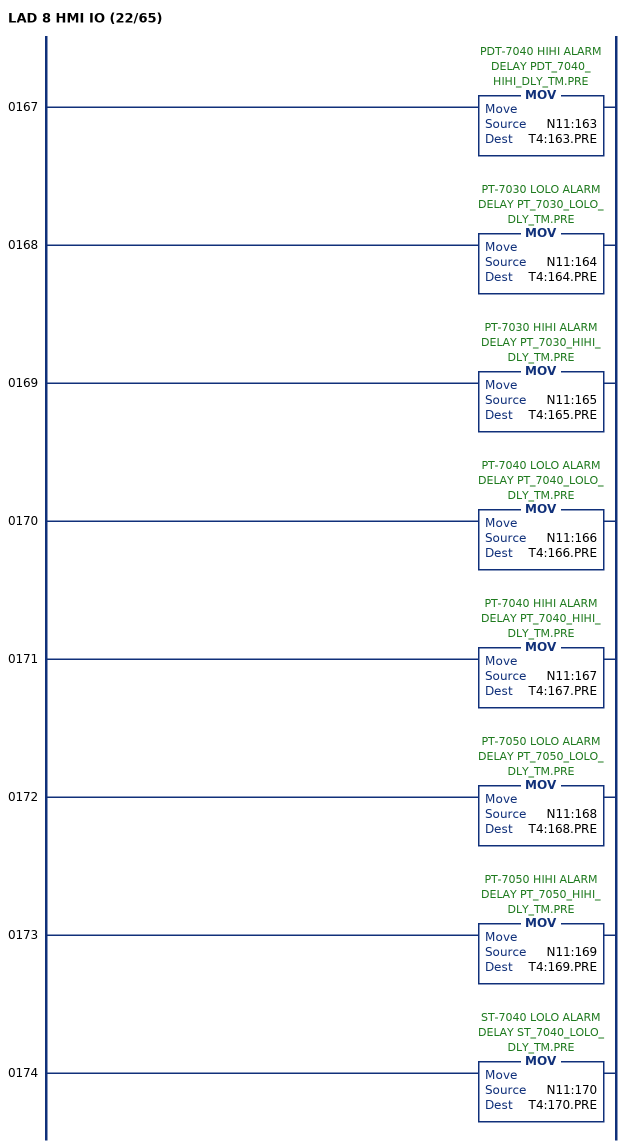
% Rung: 167 %
SOR MOV N11:163 T4:163.PRE EOR
%   N11:163  PDT_7040_HIHI_DLY_SP  "PDT-7040 HIHI ALARM DELAY SP FROM HMI" %
%   T4:163  PDT_7040_HIHI_DLY_TM  "PDT-7040 HIHI ALARM DELAY" %
% Rung: 168 %
SOR MOV N11:164 T4:164.PRE EOR
%   N11:164  PT_7030_LOLO_DLY_SP  "PT-7030 LOLO ALARM DELAY SP FROM HMI" %
%   T4:164  PT_7030_LOLO_DLY_TM  "PT-7030 LOLO ALARM DELAY" %
% Rung: 169 %
SOR MOV N11:165 T4:165.PRE EOR
%   N11:165  PT_7030_HIHI_DLY_SP  "PT-7030 HIHI ALARM DELAY SP FROM HMI" %
%   T4:165  PT_7030_HIHI_DLY_TM  "PT-7030 HIHI ALARM DELAY" %
% Rung: 170 %
SOR MOV N11:166 T4:166.PRE EOR
%   N11:166  PT_7040_LOLO_DLY_SP  "PT-7040 LOLO ALARM DELAY SP FROM HMI" %
%   T4:166  PT_7040_LOLO_DLY_TM  "PT-7040 LOLO ALARM DELAY" %
% Rung: 171 %
SOR MOV N11:167 T4:167.PRE EOR
%   N11:167  PT_7040_HIHI_DLY_SP  "PT-7040 HIHI ALARM DELAY SP FROM HMI" %
%   T4:167  PT_7040_HIHI_DLY_TM  "PT-7040 HIHI ALARM DELAY" %
% Rung: 172 %
SOR MOV N11:168 T4:168.PRE EOR
%   N11:168  PT_7050_LOLO_DLY_SP  "PT-7050 LOLO ALARM DELAY SP FROM HMI" %
%   T4:168  PT_7050_LOLO_DLY_TM  "PT-7050 LOLO ALARM DELAY" %
% Rung: 173 %
SOR MOV N11:169 T4:169.PRE EOR
%   N11:169  PT_7050_HIHI_DLY_SP  "PT-7050 HIHI ALARM DELAY SP FROM HMI" %
%   T4:169  PT_7050_HIHI_DLY_TM  "PT-7050 HIHI ALARM DELAY" %
% Rung: 174 %
SOR MOV N11:170 T4:170.PRE EOR
%   N11:170  ST_7040_LOLO_DLY_SP  "ST-7040 LOLO ALARM DELAY SP FROM HMI" %
%   T4:170  ST_7040_LOLO_DLY_TM  "ST-7040 LOLO ALARM DELAY" %

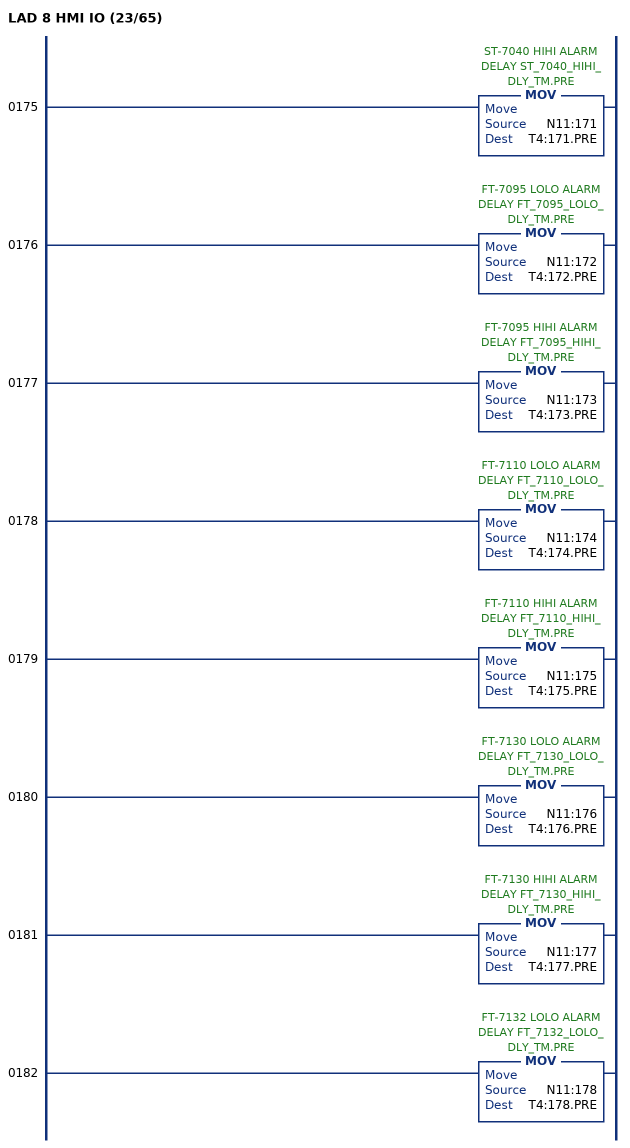
% Rung: 175 %
SOR MOV N11:171 T4:171.PRE EOR
%   N11:171  ST_7040_HIHI_DLY_SP  "ST-7040 HIHI ALARM DELAY SP FROM HMI" %
%   T4:171  ST_7040_HIHI_DLY_TM  "ST-7040 HIHI ALARM DELAY" %
% Rung: 176 %
SOR MOV N11:172 T4:172.PRE EOR
%   N11:172  FT_7095_LOLO_DLY_SP  "FT-7095 LOLO ALARM DELAY SP FROM HMI" %
%   T4:172  FT_7095_LOLO_DLY_TM  "FT-7095 LOLO ALARM DELAY" %
% Rung: 177 %
SOR MOV N11:173 T4:173.PRE EOR
%   N11:173  FT_7095_HIHI_DLY_SP  "FT-7095 HIHI ALARM DELAY SP FROM HMI" %
%   T4:173  FT_7095_HIHI_DLY_TM  "FT-7095 HIHI ALARM DELAY" %
% Rung: 178 %
SOR MOV N11:174 T4:174.PRE EOR
%   N11:174  FT_7110_LOLO_DLY_SP  "FT-7110 LOLO ALARM DELAY SP FROM HMI" %
%   T4:174  FT_7110_LOLO_DLY_TM  "FT-7110 LOLO ALARM DELAY" %
% Rung: 179 %
SOR MOV N11:175 T4:175.PRE EOR
%   N11:175  FT_7110_HIHI_DLY_SP  "FT-7110 HIHI ALARM DELAY SP FROM HMI" %
%   T4:175  FT_7110_HIHI_DLY_TM  "FT-7110 HIHI ALARM DELAY" %
% Rung: 180 %
SOR MOV N11:176 T4:176.PRE EOR
%   N11:176  FT_7130_LOLO_DLY_SP  "FT-7130 LOLO ALARM DELAY SP FROM HMI" %
%   T4:176  FT_7130_LOLO_DLY_TM  "FT-7130 LOLO ALARM DELAY" %
% Rung: 181 %
SOR MOV N11:177 T4:177.PRE EOR
%   N11:177  FT_7130_HIHI_DLY_SP  "FT-7130 HIHI ALARM DELAY SP FROM HMI" %
%   T4:177  FT_7130_HIHI_DLY_TM  "FT-7130 HIHI ALARM DELAY" %
% Rung: 182 %
SOR MOV N11:178 T4:178.PRE EOR
%   N11:178  FT_7132_LOLO_DLY_SP  "FT-7132 LOLO ALARM DELAY SP FROM HMI" %
%   T4:178  FT_7132_LOLO_DLY_TM  "FT-7132 LOLO ALARM DELAY" %

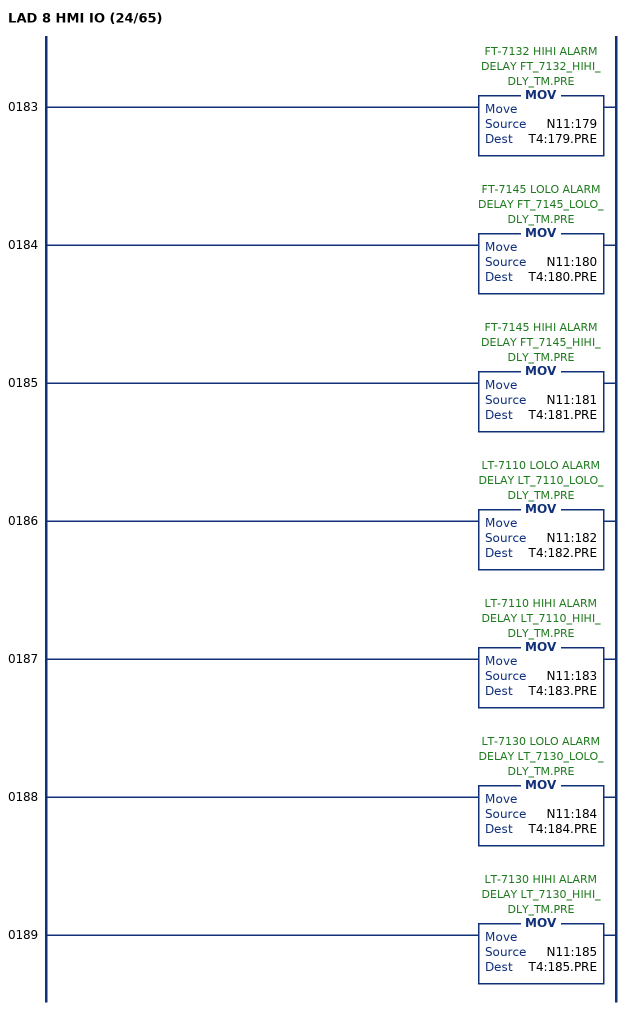
% Rung: 183 %
SOR MOV N11:179 T4:179.PRE EOR
%   N11:179  FT_7132_HIHI_DLY_SP  "FT-7132 HIHI ALARM DELAY SP FROM HMI" %
%   T4:179  FT_7132_HIHI_DLY_TM  "FT-7132 HIHI ALARM DELAY" %
% Rung: 184 %
SOR MOV N11:180 T4:180.PRE EOR
%   N11:180  FT_7145_LOLO_DLY_SP  "FT-7145 LOLO ALARM DELAY SP FROM HMI" %
%   T4:180  FT_7145_LOLO_DLY_TM  "FT-7145 LOLO ALARM DELAY" %
% Rung: 185 %
SOR MOV N11:181 T4:181.PRE EOR
%   N11:181  FT_7145_HIHI_DLY_SP  "FT-7145 HIHI ALARM DELAY SP FROM HMI" %
%   T4:181  FT_7145_HIHI_DLY_TM  "FT-7145 HIHI ALARM DELAY" %
% Rung: 186 %
SOR MOV N11:182 T4:182.PRE EOR
%   N11:182  LT_7110_LOLO_DLY_SP  "LT-7110 LOLO ALARM DELAY SP FROM HMI" %
%   T4:182  LT_7110_LOLO_DLY_TM  "LT-7110 LOLO ALARM DELAY" %
% Rung: 187 %
SOR MOV N11:183 T4:183.PRE EOR
%   N11:183  LT_7110_HIHI_DLY_SP  "LT-7110 HIHI ALARM DELAY SP FROM HMI" %
%   T4:183  LT_7110_HIHI_DLY_TM  "LT-7110 HIHI ALARM DELAY" %
% Rung: 188 %
SOR MOV N11:184 T4:184.PRE EOR
%   N11:184  LT_7130_LOLO_DLY_SP  "LT-7130 LOLO ALARM DELAY SP FROM HMI" %
%   T4:184  LT_7130_LOLO_DLY_TM  "LT-7130 LOLO ALARM DELAY" %
% Rung: 189 %
SOR MOV N11:185 T4:185.PRE EOR
%   N11:185  LT_7130_HIHI_DLY_SP  "LT-7130 HIHI ALARM DELAY SP FROM HMI" %
%   T4:185  LT_7130_HIHI_DLY_TM  "LT-7130 HIHI ALARM DELAY" %

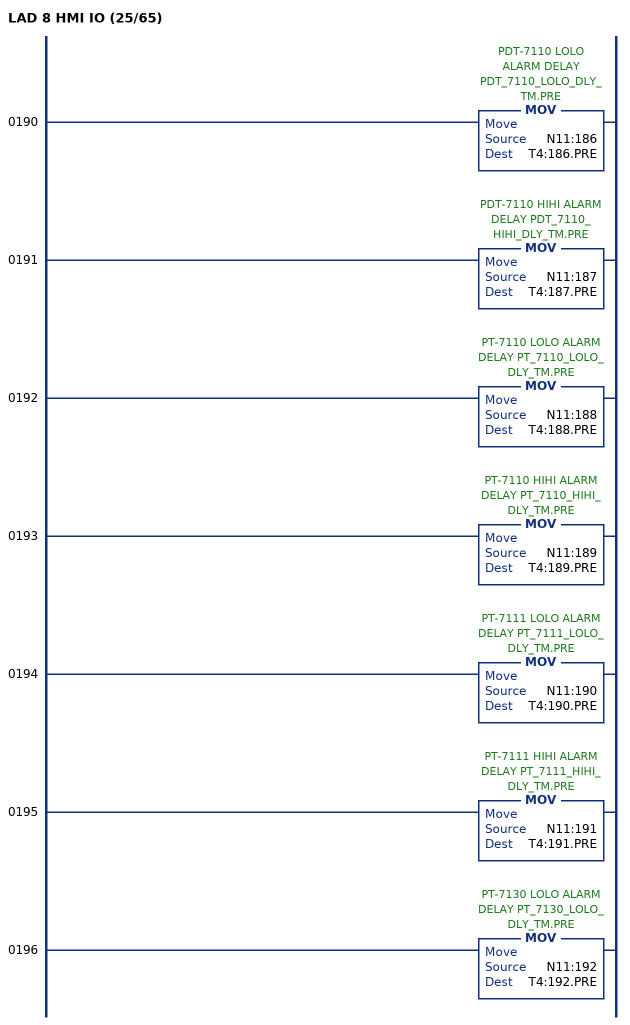
% Rung: 190 %
SOR MOV N11:186 T4:186.PRE EOR
%   N11:186  PDT_7110_LOLO_DLY_SP  "PDT-7110 LOLO ALARM DELAY SP FROM HMI" %
%   T4:186  PDT_7110_LOLO_DLY_TM  "PDT-7110 LOLO ALARM DELAY" %
% Rung: 191 %
SOR MOV N11:187 T4:187.PRE EOR
%   N11:187  PDT_7110_HIHI_DLY_SP  "PDT-7110 HIHI ALARM DELAY SP FROM HMI" %
%   T4:187  PDT_7110_HIHI_DLY_TM  "PDT-7110 HIHI ALARM DELAY" %
% Rung: 192 %
SOR MOV N11:188 T4:188.PRE EOR
%   N11:188  PT_7110_LOLO_DLY_SP  "PT-7110 LOLO ALARM DELAY SP FROM HMI" %
%   T4:188  PT_7110_LOLO_DLY_TM  "PT-7110 LOLO ALARM DELAY" %
% Rung: 193 %
SOR MOV N11:189 T4:189.PRE EOR
%   N11:189  PT_7110_HIHI_DLY_SP  "PT-7110 HIHI ALARM DELAY SP FROM HMI" %
%   T4:189  PT_7110_HIHI_DLY_TM  "PT-7110 HIHI ALARM DELAY" %
% Rung: 194 %
SOR MOV N11:190 T4:190.PRE EOR
%   N11:190  PT_7111_LOLO_DLY_SP  "PT-7111 LOLO ALARM DELAY SP FROM HMI" %
%   T4:190  PT_7111_LOLO_DLY_TM  "PT-7111 LOLO ALARM DELAY" %
% Rung: 195 %
SOR MOV N11:191 T4:191.PRE EOR
%   N11:191  PT_7111_HIHI_DLY_SP  "PT-7111 HIHI ALARM DELAY SP FROM HMI" %
%   T4:191  PT_7111_HIHI_DLY_TM  "PT-7111 HIHI ALARM DELAY" %
% Rung: 196 %
SOR MOV N11:192 T4:192.PRE EOR
%   N11:192  PT_7130_LOLO_DLY_SP  "PT-7130 LOLO ALARM DELAY SP FROM HMI" %
%   T4:192  PT_7130_LOLO_DLY_TM  "PT-7130 LOLO ALARM DELAY" %

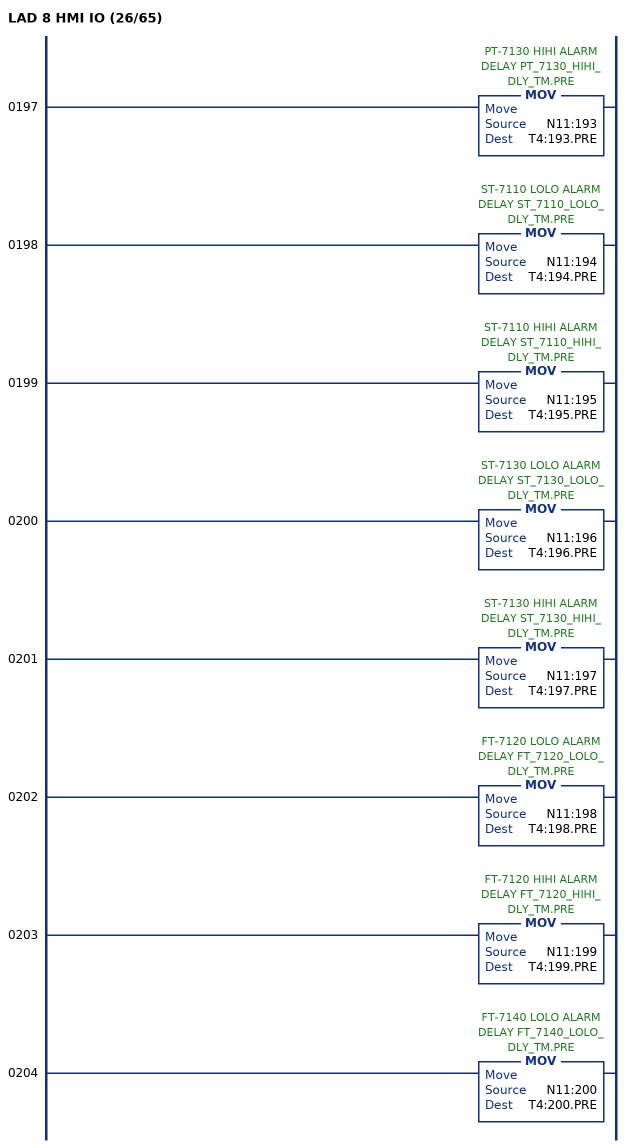
% Rung: 197 %
SOR MOV N11:193 T4:193.PRE EOR
%   N11:193  PT_7130_HIHI_DLY_SP  "PT-7130 HIHI ALARM DELAY SP FROM HMI" %
%   T4:193  PT_7130_HIHI_DLY_TM  "PT-7130 HIHI ALARM DELAY" %
% Rung: 198 %
SOR MOV N11:194 T4:194.PRE EOR
%   N11:194  ST_7110_LOLO_DLY_SP  "ST-7110 LOLO ALARM DELAY SP FROM HMI" %
%   T4:194  ST_7110_LOLO_DLY_TM  "ST-7110 LOLO ALARM DELAY" %
% Rung: 199 %
SOR MOV N11:195 T4:195.PRE EOR
%   N11:195  ST_7110_HIHI_DLY_SP  "ST-7110 HIHI ALARM DELAY SP FROM HMI" %
%   T4:195  ST_7110_HIHI_DLY_TM  "ST-7110 HIHI ALARM DELAY" %
% Rung: 200 %
SOR MOV N11:196 T4:196.PRE EOR
%   N11:196  ST_7130_LOLO_DLY_SP  "ST-7130 LOLO ALARM DELAY SP FROM HMI" %
%   T4:196  ST_7130_LOLO_DLY_TM  "ST-7130 LOLO ALARM DELAY" %
% Rung: 201 %
SOR MOV N11:197 T4:197.PRE EOR
%   N11:197  ST_7130_HIHI_DLY_SP  "ST-7130 HIHI ALARM DELAY SP FROM HMI" %
%   T4:197  ST_7130_HIHI_DLY_TM  "ST-7130 HIHI ALARM DELAY" %
% Rung: 202 %
SOR MOV N11:198 T4:198.PRE EOR
%   N11:198  FT_7120_LOLO_DLY_SP  "FT-7120 LOLO ALARM DELAY SP FROM HMI" %
%   T4:198  FT_7120_LOLO_DLY_TM  "FT-7120 LOLO ALARM DELAY" %
% Rung: 203 %
SOR MOV N11:199 T4:199.PRE EOR
%   N11:199  FT_7120_HIHI_DLY_SP  "FT-7120 HIHI ALARM DELAY SP FROM HMI" %
%   T4:199  FT_7120_HIHI_DLY_TM  "FT-7120 HIHI ALARM DELAY" %
% Rung: 204 %
SOR MOV N11:200 T4:200.PRE EOR
%   N11:200  FT_7140_LOLO_DLY_SP  "FT-7140 LOLO ALARM DELAY SP FROM HMI" %
%   T4:200  FT_7140_LOLO_DLY_TM  "FT-7140 LOLO ALARM DELAY" %

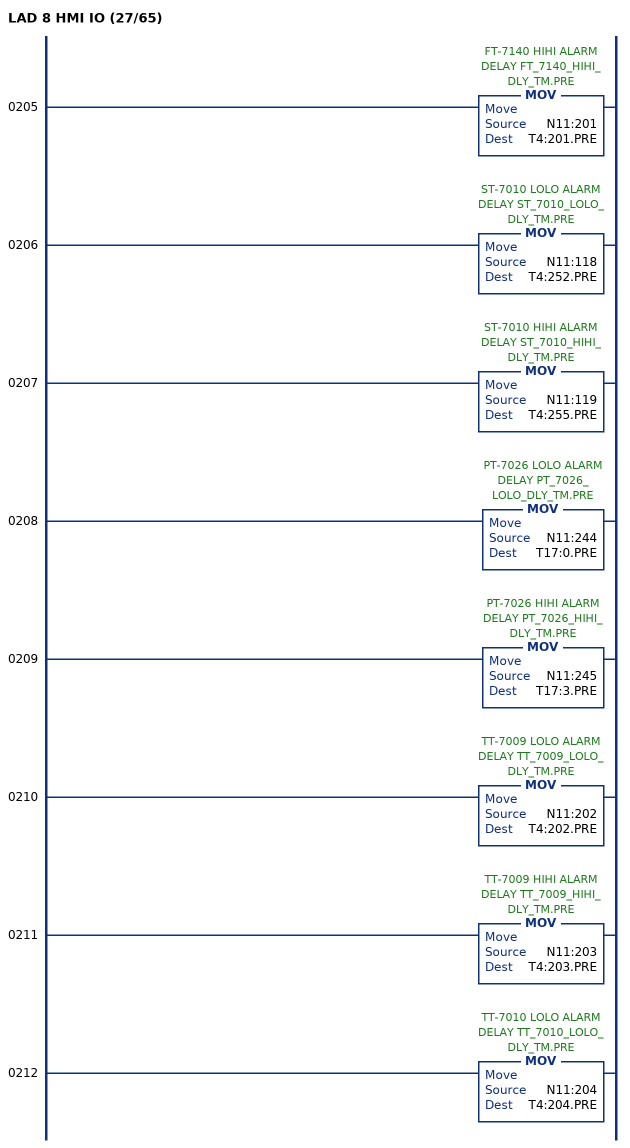
% Rung: 205 %
SOR MOV N11:201 T4:201.PRE EOR
%   N11:201  FT_7140_HIHI_DLY_SP  "FT-7140 HIHI ALARM DELAY SP FROM HMI" %
%   T4:201  FT_7140_HIHI_DLY_TM  "FT-7140 HIHI ALARM DELAY" %
% Rung: 206 %
SOR MOV N11:118 T4:252.PRE EOR
%   N11:118  ST_7010_LOLO_DLY_SP  "ST-7010 LL ALARM DELAY SP FROM HMI" %
%   T4:252  ST_7010_LOLO_DLY_TM  "ST-7010 LOLO ALARM DELAY" %
% Rung: 207 %
SOR MOV N11:119 T4:255.PRE EOR
%   N11:119  ST_7010_HIHI_DLY_SP  "ST-7010 HH ALARM DELAY SP FROM HMI" %
%   T4:255  ST_7010_HIHI_DLY_TM  "ST-7010 HIHI ALARM DELAY" %
% Rung: 208 %
SOR MOV N11:244 T17:0.PRE EOR
%   N11:244  PT_7026_LOLO_DLY_SP  "PT-7026 LL ALARM DELAY SP FROM HMI" %
%   T17:0  PT_7026_LOLO_DLY_TM  "PT-7026 LOLO ALARM DELAY" %
% Rung: 209 %
SOR MOV N11:245 T17:3.PRE EOR
%   N11:245  PT_7026_HIHI_DLY_SP  "PT-7026 HH ALARM DELAY SP FROM HMI" %
%   T17:3  PT_7026_HIHI_DLY_TM  "PT-7026 HIHI ALARM DELAY" %
% Rung: 210 %
SOR MOV N11:202 T4:202.PRE EOR
%   N11:202  TT_7009_LOLO_DLY_SP  "TT-7009 LOLO ALARM DELAY SP FROM HMI" %
%   T4:202  TT_7009_LOLO_DLY_TM  "TT-7009 LOLO ALARM DELAY" %
% Rung: 211 %
SOR MOV N11:203 T4:203.PRE EOR
%   N11:203  TT_7009_HIHI_DLY_SP  "TT-7009 HIHI ALARM DELAY SP FROM HMI" %
%   T4:203  TT_7009_HIHI_DLY_TM  "TT-7009 HIHI ALARM DELAY" %
% Rung: 212 %
SOR MOV N11:204 T4:204.PRE EOR
%   N11:204  TT_7010_LOLO_DLY_SP  "TT-7010 LOLO ALARM DELAY SP FROM HMI" %
%   T4:204  TT_7010_LOLO_DLY_TM  "TT-7010 LOLO ALARM DELAY" %

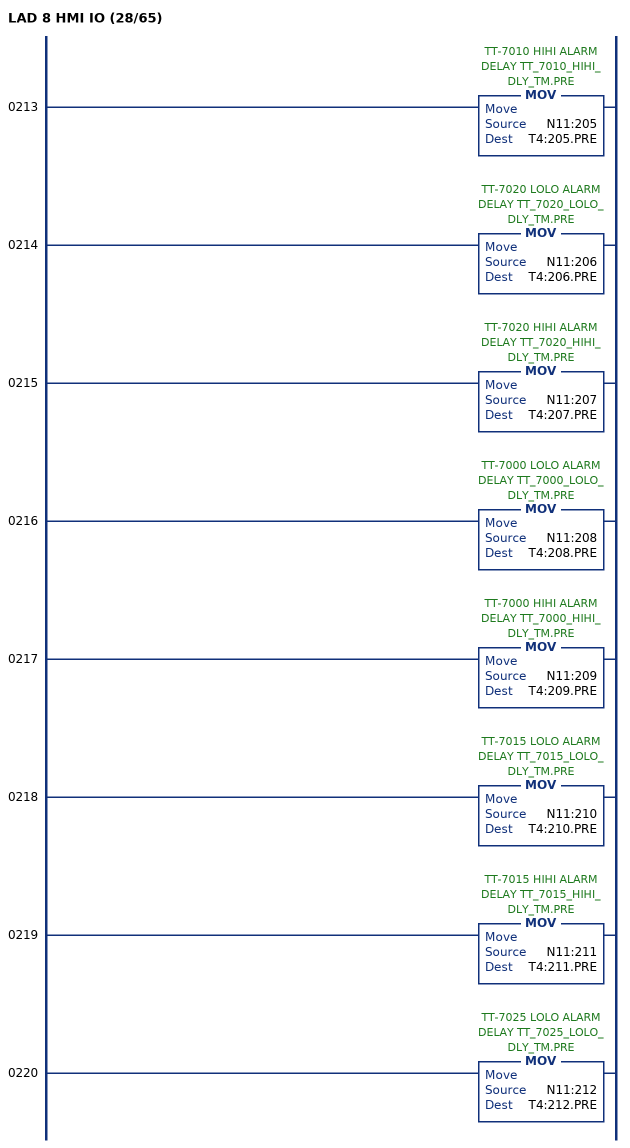
% Rung: 213 %
SOR MOV N11:205 T4:205.PRE EOR
%   N11:205  TT_7010_HIHI_DLY_SP  "TT-7010 HIHI ALARM DELAY SP FROM HMI" %
%   T4:205  TT_7010_HIHI_DLY_TM  "TT-7010 HIHI ALARM DELAY" %
% Rung: 214 %
SOR MOV N11:206 T4:206.PRE EOR
%   N11:206  TT_7020_LOLO_DLY_SP  "TT-7020 LOLO ALARM DELAY SP FROM HMI" %
%   T4:206  TT_7020_LOLO_DLY_TM  "TT-7020 LOLO ALARM DELAY" %
% Rung: 215 %
SOR MOV N11:207 T4:207.PRE EOR
%   N11:207  TT_7020_HIHI_DLY_SP  "TT-7020 HIHI ALARM DELAY SP FROM HMI" %
%   T4:207  TT_7020_HIHI_DLY_TM  "TT-7020 HIHI ALARM DELAY" %
% Rung: 216 %
SOR MOV N11:208 T4:208.PRE EOR
%   N11:208  TT_7000_LOLO_DLY_SP  "TT-7000 LOLO ALARM DELAY SP FROM HMI" %
%   T4:208  TT_7000_LOLO_DLY_TM  "TT-7000 LOLO ALARM DELAY" %
% Rung: 217 %
SOR MOV N11:209 T4:209.PRE EOR
%   N11:209  TT_7000_HIHI_DLY_SP  "TT-7000 HIHI ALARM DELAY SP FROM HMI" %
%   T4:209  TT_7000_HIHI_DLY_TM  "TT-7000 HIHI ALARM DELAY" %
% Rung: 218 %
SOR MOV N11:210 T4:210.PRE EOR
%   N11:210  TT_7015_LOLO_DLY_SP  "TT-7015 LOLO ALARM DELAY SP FROM HMI" %
%   T4:210  TT_7015_LOLO_DLY_TM  "TT-7015 LOLO ALARM DELAY" %
% Rung: 219 %
SOR MOV N11:211 T4:211.PRE EOR
%   N11:211  TT_7015_HIHI_DLY_SP  "TT-7015 HIHI ALARM DELAY SP FROM HMI" %
%   T4:211  TT_7015_HIHI_DLY_TM  "TT-7015 HIHI ALARM DELAY" %
% Rung: 220 %
SOR MOV N11:212 T4:212.PRE EOR
%   N11:212  TT_7025_LOLO_DLY_SP  "TT-7025 LOLO ALARM DELAY SP FROM HMI" %
%   T4:212  TT_7025_LOLO_DLY_TM  "TT-7025 LOLO ALARM DELAY" %

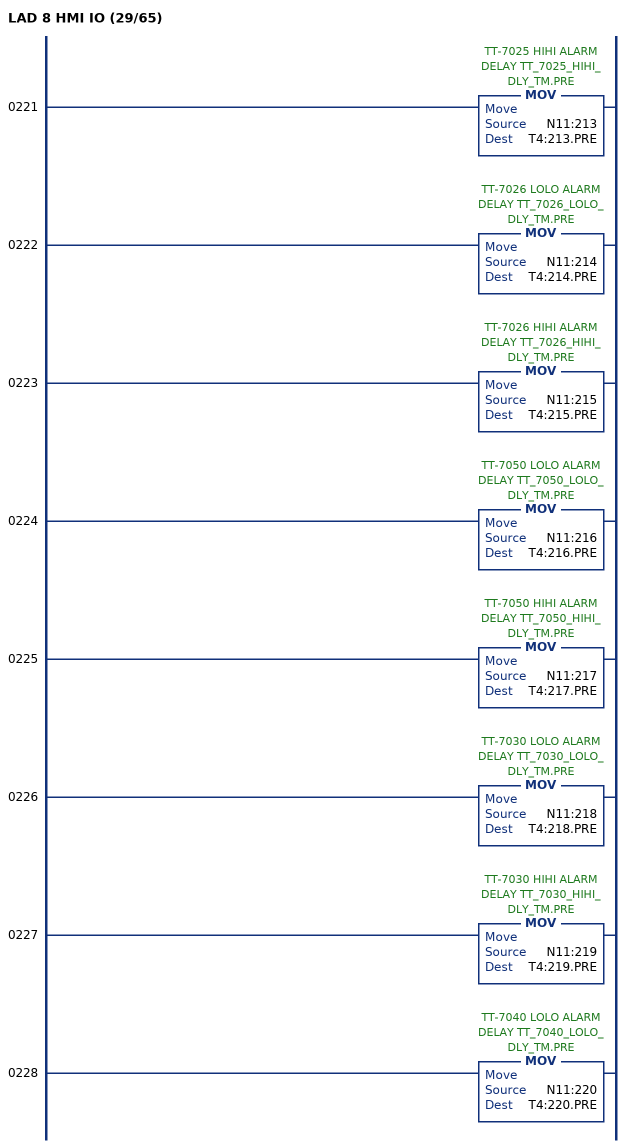
% Rung: 221 %
SOR MOV N11:213 T4:213.PRE EOR
%   N11:213  TT_7025_HIHIDLY_SP  "TT-7025 HIHI ALARM DELAY SP FROM HMI" %
%   T4:213  TT_7025_HIHI_DLY_TM  "TT-7025 HIHI ALARM DELAY" %
% Rung: 222 %
SOR MOV N11:214 T4:214.PRE EOR
%   N11:214  TT_7026_LOLO_DLY_SP  "TT-7026 LOLO ALARM DELAY SP FROM HMI" %
%   T4:214  TT_7026_LOLO_DLY_TM  "TT-7026 LOLO ALARM DELAY" %
% Rung: 223 %
SOR MOV N11:215 T4:215.PRE EOR
%   N11:215  TT_7026_HIHI_DLY_SP  "TT-7026 HIHI ALARM DELAY SP FROM HMI" %
%   T4:215  TT_7026_HIHI_DLY_TM  "TT-7026 HIHI ALARM DELAY" %
% Rung: 224 %
SOR MOV N11:216 T4:216.PRE EOR
%   N11:216  TT_7050_LOLO_DLY_SP  "TT-7050 LOLO ALARM DELAY SP FROM HMI" %
%   T4:216  TT_7050_LOLO_DLY_TM  "TT-7050 LOLO ALARM DELAY" %
% Rung: 225 %
SOR MOV N11:217 T4:217.PRE EOR
%   N11:217  TT_7050_HIHI_DLY_SP  "TT-7050 HIHI ALARM DELAY SP FROM HMI" %
%   T4:217  TT_7050_HIHI_DLY_TM  "TT-7050 HIHI ALARM DELAY" %
% Rung: 226 %
SOR MOV N11:218 T4:218.PRE EOR
%   N11:218  TT_7030_LOLO_DLY_SP  "TT-7030 LOLO ALARM DELAY SP FROM HMI" %
%   T4:218  TT_7030_LOLO_DLY_TM  "TT-7030 LOLO ALARM DELAY" %
% Rung: 227 %
SOR MOV N11:219 T4:219.PRE EOR
%   N11:219  TT_7030_HIHI_DLY_SP  "TT-7030 HIHI ALARM DELAY SP FROM HMI" %
%   T4:219  TT_7030_HIHI_DLY_TM  "TT-7030 HIHI ALARM DELAY" %
% Rung: 228 %
SOR MOV N11:220 T4:220.PRE EOR
%   N11:220  TT_7040_LOLO_DLY_SP  "TT-7040 LOLO ALARM DELAY SP FROM HMI" %
%   T4:220  TT_7040_LOLO_DLY_TM  "TT-7040 LOLO ALARM DELAY" %

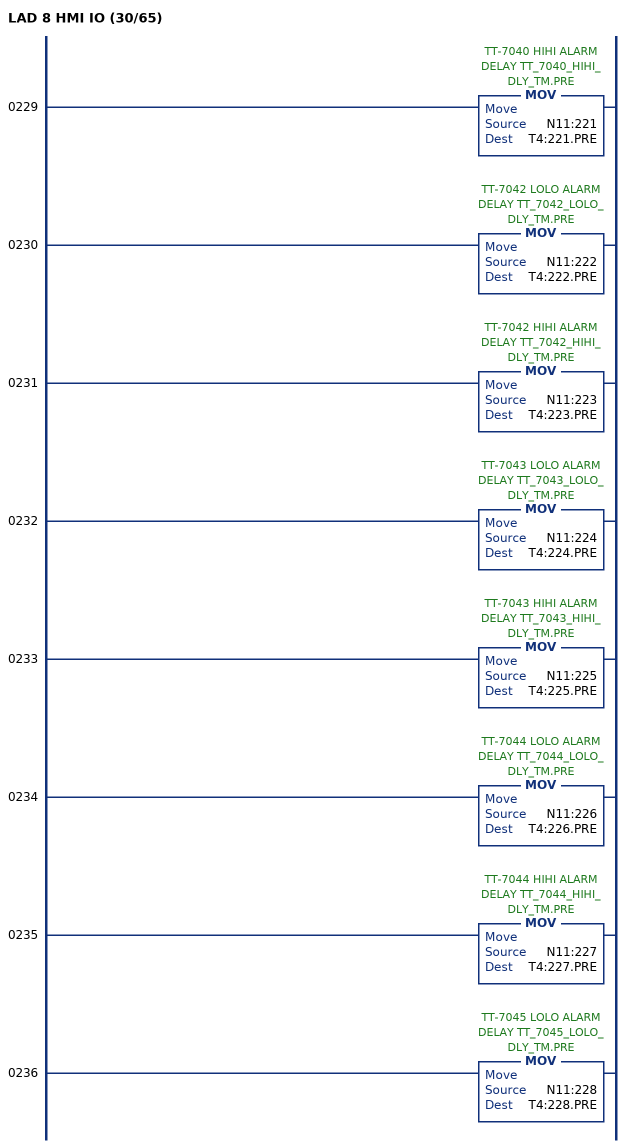
% Rung: 229 %
SOR MOV N11:221 T4:221.PRE EOR
%   N11:221  TT_7040_HIHI_DLY_SP  "TT-7040 HIHI ALARM DELAY SP FROM HMI" %
%   T4:221  TT_7040_HIHI_DLY_TM  "TT-7040 HIHI ALARM DELAY" %
% Rung: 230 %
SOR MOV N11:222 T4:222.PRE EOR
%   N11:222  TT_7042_LOLO_DLY_SP  "TT-7042 LOLO ALARM DELAY SP FROM HMI" %
%   T4:222  TT_7042_LOLO_DLY_TM  "TT-7042 LOLO ALARM DELAY" %
% Rung: 231 %
SOR MOV N11:223 T4:223.PRE EOR
%   N11:223  TT_7042_HIHI_DLY_SP  "TT-7042 HIHI ALARM DELAY SP FROM HMI" %
%   T4:223  TT_7042_HIHI_DLY_TM  "TT-7042 HIHI ALARM DELAY" %
% Rung: 232 %
SOR MOV N11:224 T4:224.PRE EOR
%   N11:224  TT_7043_LOLO_DLY_SP  "TT-7043 LOLO ALARM DELAY SP FROM HMI" %
%   T4:224  TT_7043_LOLO_DLY_TM  "TT-7043 LOLO ALARM DELAY" %
% Rung: 233 %
SOR MOV N11:225 T4:225.PRE EOR
%   N11:225  TT_7043_HIHI_DLY_SP  "TT-7043 HIHI ALARM DELAY SP FROM HMI" %
%   T4:225  TT_7043_HIHI_DLY_TM  "TT-7043 HIHI ALARM DELAY" %
% Rung: 234 %
SOR MOV N11:226 T4:226.PRE EOR
%   N11:226  TT_7044_LOLO_DLY_SP  "TT-7044 LOLO ALARM DELAY SP FROM HMI" %
%   T4:226  TT_7044_LOLO_DLY_TM  "TT-7044 LOLO ALARM DELAY" %
% Rung: 235 %
SOR MOV N11:227 T4:227.PRE EOR
%   N11:227  TT_7044_HIHI_DLY_SP  "TT-7044 HIHI ALARM DELAY SP FROM HMI" %
%   T4:227  TT_7044_HIHI_DLY_TM  "TT-7044 HIHI ALARM DELAY" %
% Rung: 236 %
SOR MOV N11:228 T4:228.PRE EOR
%   N11:228  TT_7045_LOLO_DLY_SP  "TT-7045 LOLO ALARM DELAY SP FROM HMI" %
%   T4:228  TT_7045_LOLO_DLY_TM  "TT-7045 LOLO ALARM DELAY" %

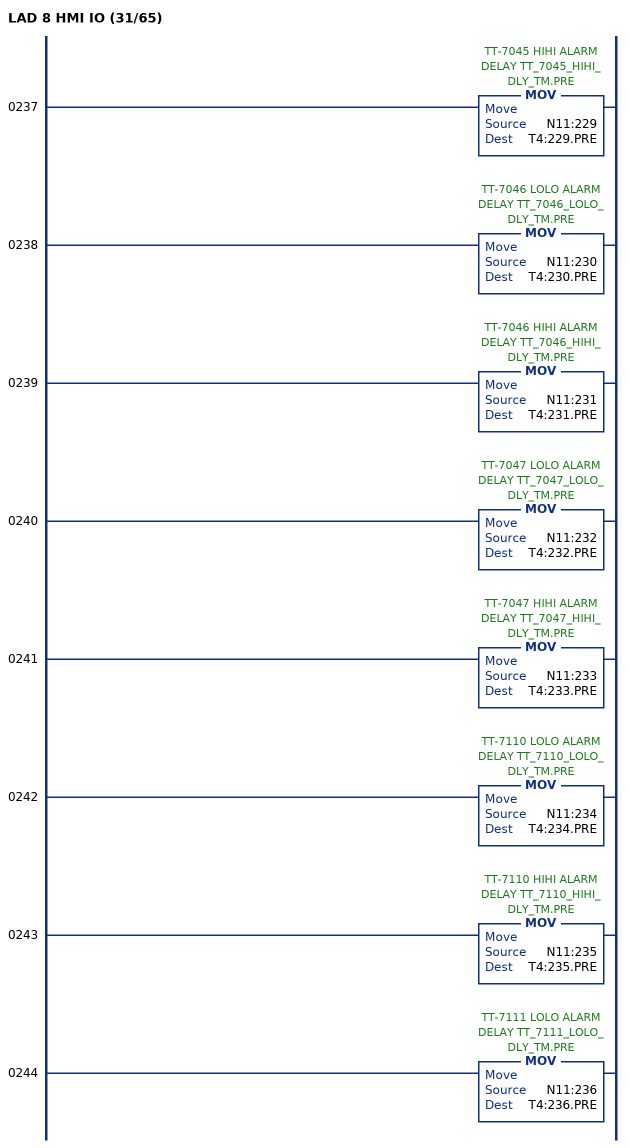
% Rung: 237 %
SOR MOV N11:229 T4:229.PRE EOR
%   N11:229  TT_7045_HIHI_DLY_SP  "TT-7045 HIHI ALARM DELAY SP FROM HMI" %
%   T4:229  TT_7045_HIHI_DLY_TM  "TT-7045 HIHI ALARM DELAY" %
% Rung: 238 %
SOR MOV N11:230 T4:230.PRE EOR
%   N11:230  TT_7046_LOLO_DLY_SP  "TT-7046 LOLO ALARM DELAY SP FROM HMI" %
%   T4:230  TT_7046_LOLO_DLY_TM  "TT-7046 LOLO ALARM DELAY" %
% Rung: 239 %
SOR MOV N11:231 T4:231.PRE EOR
%   N11:231  TT_7046_HIHI_DLY_SP  "TT-7046 HIHI ALARM DELAY SP FROM HMI" %
%   T4:231  TT_7046_HIHI_DLY_TM  "TT-7046 HIHI ALARM DELAY" %
% Rung: 240 %
SOR MOV N11:232 T4:232.PRE EOR
%   N11:232  TT_7047_LOLO_DLY_SP  "TT-7047 LOLO ALARM DELAY SP FROM HMI" %
%   T4:232  TT_7047_LOLO_DLY_TM  "TT-7047 LOLO ALARM DELAY" %
% Rung: 241 %
SOR MOV N11:233 T4:233.PRE EOR
%   N11:233  TT_7047_HIHI_DLY_SP  "TT-7047 HIHI ALARM DELAY SP FROM HMI" %
%   T4:233  TT_7047_HIHI_DLY_TM  "TT-7047 HIHI ALARM DELAY" %
% Rung: 242 %
SOR MOV N11:234 T4:234.PRE EOR
%   N11:234  TT_7110_LOLO_DLY_SP  "TT-7110 LOLO ALARM DELAY SP FROM HMI" %
%   T4:234  TT_7110_LOLO_DLY_TM  "TT-7110 LOLO ALARM DELAY" %
% Rung: 243 %
SOR MOV N11:235 T4:235.PRE EOR
%   N11:235  TT_7110_HIHI_DLY_SP  "TT-7110 HIHI ALARM DELAY SP FROM HMI" %
%   T4:235  TT_7110_HIHI_DLY_TM  "TT-7110 HIHI ALARM DELAY" %
% Rung: 244 %
SOR MOV N11:236 T4:236.PRE EOR
%   N11:236  TT_7111_LOLO_DLY_SP  "TT-7111 LOLO ALARM DELAY SP FROM HMI" %
%   T4:236  TT_7111_LOLO_DLY_TM  "TT-7111 LOLO ALARM DELAY" %

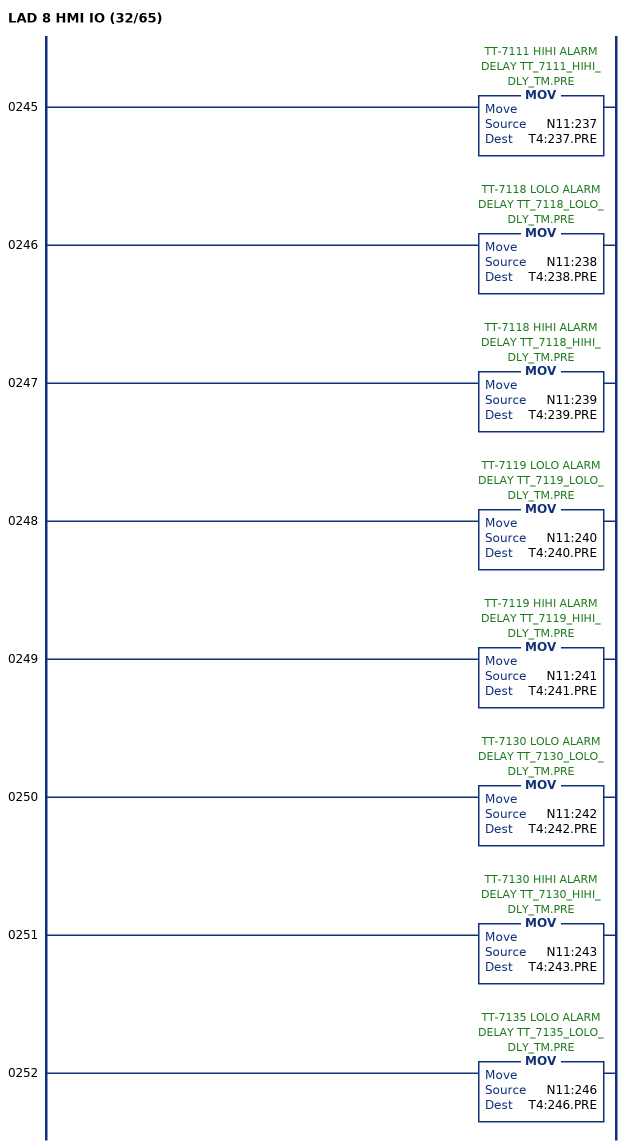
% Rung: 245 %
SOR MOV N11:237 T4:237.PRE EOR
%   N11:237  TT_7111_HIHI_DLY_SP  "TT-7111 HIHI ALARM DELAY SP FROM HMI" %
%   T4:237  TT_7111_HIHI_DLY_TM  "TT-7111 HIHI ALARM DELAY" %
% Rung: 246 %
SOR MOV N11:238 T4:238.PRE EOR
%   N11:238  TT_7118_LOLO_DLY_SP  "TT-7118 LOLO ALARM DELAY SP FROM HMI" %
%   T4:238  TT_7118_LOLO_DLY_TM  "TT-7118 LOLO ALARM DELAY" %
% Rung: 247 %
SOR MOV N11:239 T4:239.PRE EOR
%   N11:239  TT_7118_HIHI_DLY_SP  "TT-7118 HIHI ALARM DELAY SP FROM HMI" %
%   T4:239  TT_7118_HIHI_DLY_TM  "TT-7118 HIHI ALARM DELAY" %
% Rung: 248 %
SOR MOV N11:240 T4:240.PRE EOR
%   N11:240  TT_7119_LOLO_DLY_SP  "TT-7119 LOLO ALARM DELAY SP FROM HMI" %
%   T4:240  TT_7119_LOLO_DLY_TM  "TT-7119 LOLO ALARM DELAY" %
% Rung: 249 %
SOR MOV N11:241 T4:241.PRE EOR
%   N11:241  TT_7119_HIHI_DLY_SP  "TT-7119 HIHI ALARM DELAY SP FROM HMI" %
%   T4:241  TT_7119_HIHI_DLY_TM  "TT-7119 HIHI ALARM DELAY" %
% Rung: 250 %
SOR MOV N11:242 T4:242.PRE EOR
%   N11:242  TT_7130_LOLO_DLY_SP  "TT-7130 LOLO ALARM DELAY SP FROM HMI" %
%   T4:242  TT_7130_LOLO_DLY_TM  "TT-7130 LOLO ALARM DELAY" %
% Rung: 251 %
SOR MOV N11:243 T4:243.PRE EOR
%   N11:243  TT_7130_HIHI_DLY_SP  "TT-7130 HIHI ALARM DELAY SP FROM HMI" %
%   T4:243  TT_7130_HIHI_DLY_TM  "TT-7130 HIHI ALARM DELAY" %
% Rung: 252 %
SOR MOV N11:246 T4:246.PRE EOR
%   N11:246  TT_7135_LOLO_DLY_SP  "TT-7135 LOLO ALARM DELAY SP FROM HMI" %
%   T4:246  TT_7135_LOLO_DLY_TM  "TT-7135 LOLO ALARM DELAY" %

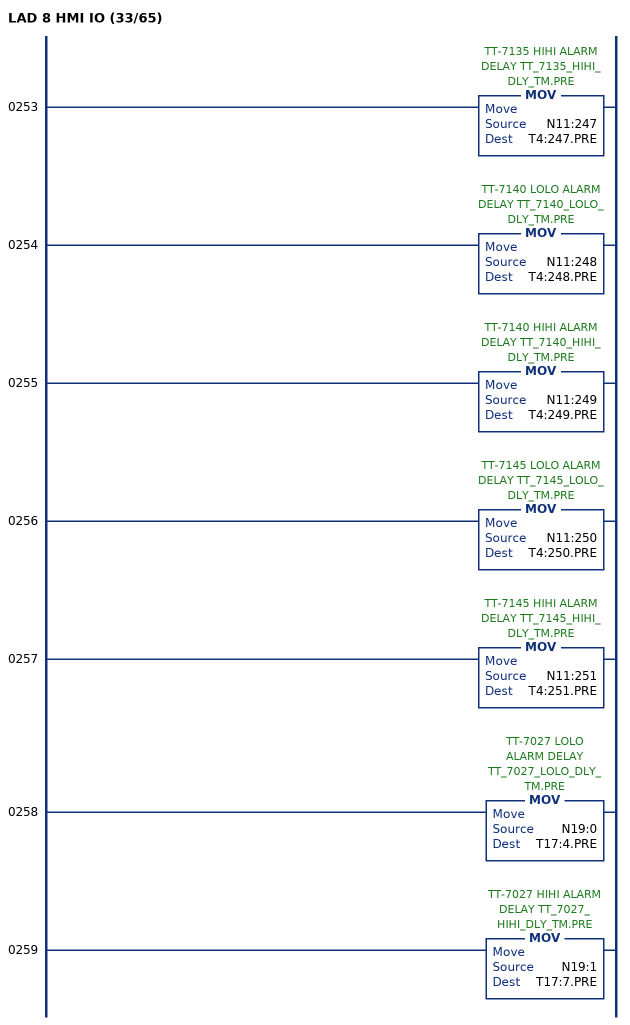
% Rung: 253 %
SOR MOV N11:247 T4:247.PRE EOR
%   N11:247  TT_7135_HIHI_DLY_SP  "TT-7135 HIHI ALARM DELAY SP FROM HMI" %
%   T4:247  TT_7135_HIHI_DLY_TM  "TT-7135 HIHI ALARM DELAY" %
% Rung: 254 %
SOR MOV N11:248 T4:248.PRE EOR
%   N11:248  TT_7140_LOLO_DLY_SP  "TT-7140 LOLO ALARM DELAY SP FROM HMI" %
%   T4:248  TT_7140_LOLO_DLY_TM  "TT-7140 LOLO ALARM DELAY" %
% Rung: 255 %
SOR MOV N11:249 T4:249.PRE EOR
%   N11:249  TT_7140_HIHI_DLY_SP  "TT-7140 HIHI ALARM DELAY SP FROM HMI" %
%   T4:249  TT_7140_HIHI_DLY_TM  "TT-7140 HIHI ALARM DELAY" %
% Rung: 256 %
SOR MOV N11:250 T4:250.PRE EOR
%   N11:250  TT_7145_LOLO_DLY_SP  "TT-7145 LOLO ALARM DELAY SP FROM HMI" %
%   T4:250  TT_7145_LOLO_DLY_TM  "TT-7145 LOLO ALARM DELAY" %
% Rung: 257 %
SOR MOV N11:251 T4:251.PRE EOR
%   N11:251  TT_7145_HIHI_DLY_SP  "TT-7145 HIHI ALARM DELAY SP FROM HMI" %
%   T4:251  TT_7145_HIHI_DLY_TM  "TT-7145 HIHI ALARM DELAY" %
% Rung: 258 %
SOR MOV N19:0 T17:4.PRE EOR
%   N19:0  TT_7027_LOLO_DLY_SP  "TT-7027 LOLO ALARM DELAY SP FROM HMI" %
%   T17:4  TT_7027_LOLO_DLY_TM  "TT-7027 LOLO ALARM DELAY" %
% Rung: 259 %
SOR MOV N19:1 T17:7.PRE EOR
%   N19:1  TT_7027_HIHI_DLY_SP  "TT-7027 HIHI ALARM DELAY SP FROM HMI" %
%   T17:7  TT_7027_HIHI_DLY_TM  "TT-7027 HIHI ALARM DELAY" %

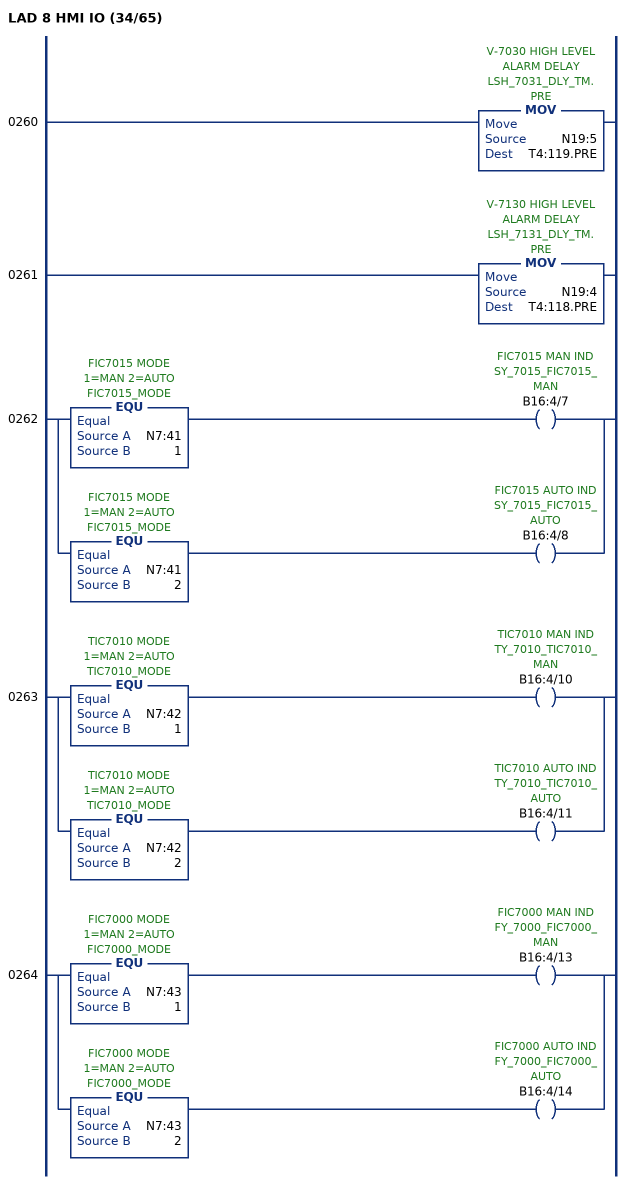
% Rung: 260 %
SOR MOV N19:5 T4:119.PRE EOR
%   N19:5  LSH_7031_DLY_SP  "LSH-7031 HIGH LEVEL ALARM DELAY SP FROM HMI" %
%   T4:119  LSH_7031_DLY_TM  "V-7030 HIGH LEVEL ALARM DELAY" %
% Rung: 261 %
SOR MOV N19:4 T4:118.PRE EOR
%   N19:4  LSH_7131_DLY_SP  "LSH-7130 HIGH LEVEL ALARM DELAY SP FROM HMI" %
%   T4:118  LSH_7131_DLY_TM  "V-7130 HIGH LEVEL ALARM DELAY" %
% Rung: 262 %
SOR BST EQU N7:41 1 OTE B16:4/7 NXB EQU N7:41 2 OTE B16:4/8 BND EOR
%   N7:41  FIC7015_MODE  "FIC7015 MODE 1=MAN 2=AUTO" %
%   B16:4/7  SY_7015_FIC7015_MAN  "FIC7015 MAN IND" %
%   B16:4/8  SY_7015_FIC7015_AUTO  "FIC7015 AUTO IND" %
% Rung: 263 %
SOR BST EQU N7:42 1 OTE B16:4/10 NXB EQU N7:42 2 OTE B16:4/11 BND EOR
%   N7:42  TIC7010_MODE  "TIC7010 MODE 1=MAN 2=AUTO" %
%   B16:4/10  TY_7010_TIC7010_MAN  "TIC7010 MAN IND" %
%   B16:4/11  TY_7010_TIC7010_AUTO  "TIC7010 AUTO IND" %
% Rung: 264 %
SOR BST EQU N7:43 1 OTE B16:4/13 NXB EQU N7:43 2 OTE B16:4/14 BND EOR
%   N7:43  FIC7000_MODE  "FIC7000 MODE 1=MAN 2=AUTO" %
%   B16:4/13  FY_7000_FIC7000_MAN  "FIC7000 MAN IND" %
%   B16:4/14  FY_7000_FIC7000_AUTO  "FIC7000 AUTO IND" %

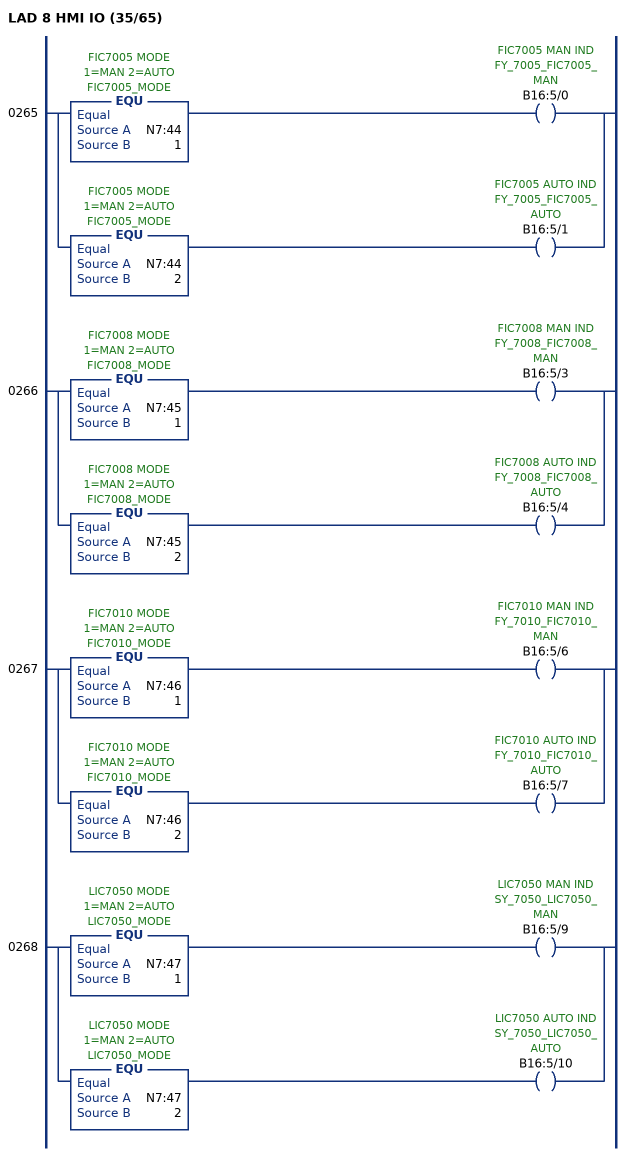
% Rung: 265 %
SOR BST EQU N7:44 1 OTE B16:5/0 NXB EQU N7:44 2 OTE B16:5/1 BND EOR
%   N7:44  FIC7005_MODE  "FIC7005 MODE 1=MAN 2=AUTO" %
%   B16:5/0  FY_7005_FIC7005_MAN  "FIC7005 MAN IND" %
%   B16:5/1  FY_7005_FIC7005_AUTO  "FIC7005 AUTO IND" %
% Rung: 266 %
SOR BST EQU N7:45 1 OTE B16:5/3 NXB EQU N7:45 2 OTE B16:5/4 BND EOR
%   N7:45  FIC7008_MODE  "FIC7008 MODE 1=MAN 2=AUTO" %
%   B16:5/3  FY_7008_FIC7008_MAN  "FIC7008 MAN IND" %
%   B16:5/4  FY_7008_FIC7008_AUTO  "FIC7008 AUTO IND" %
% Rung: 267 %
SOR BST EQU N7:46 1 OTE B16:5/6 NXB EQU N7:46 2 OTE B16:5/7 BND EOR
%   N7:46  FIC7010_MODE  "FIC7010 MODE 1=MAN 2=AUTO" %
%   B16:5/6  FY_7010_FIC7010_MAN  "FIC7010 MAN IND" %
%   B16:5/7  FY_7010_FIC7010_AUTO  "FIC7010 AUTO IND" %
% Rung: 268 %
SOR BST EQU N7:47 1 OTE B16:5/9 NXB EQU N7:47 2 OTE B16:5/10 BND EOR
%   N7:47  LIC7050_MODE  "LIC7050 MODE 1=MAN 2=AUTO" %
%   B16:5/9  SY_7050_LIC7050_MAN  "LIC7050 MAN IND" %
%   B16:5/10  SY_7050_LIC7050_AUTO  "LIC7050 AUTO IND" %

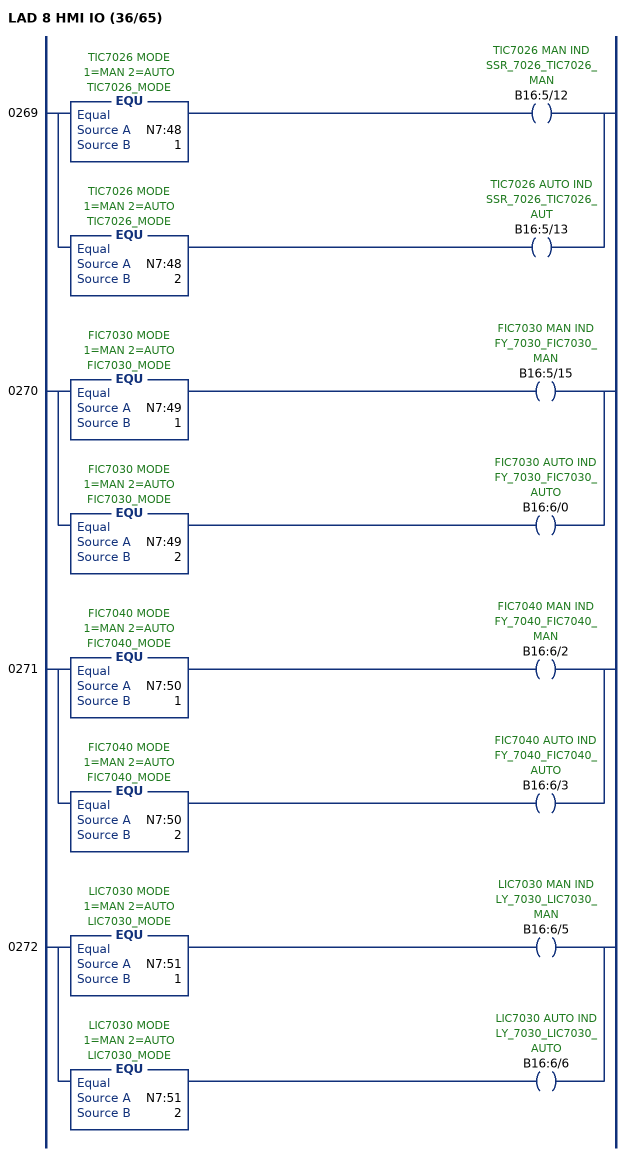
% Rung: 269 %
SOR BST EQU N7:48 1 OTE B16:5/12 NXB EQU N7:48 2 OTE B16:5/13 BND EOR
%   N7:48  TIC7026_MODE  "TIC7026 MODE 1=MAN 2=AUTO" %
%   B16:5/12  SSR_7026_TIC7026_MAN  "TIC7026 MAN IND" %
%   B16:5/13  SSR_7026_TIC7026_AUT  "TIC7026 AUTO IND" %
% Rung: 270 %
SOR BST EQU N7:49 1 OTE B16:5/15 NXB EQU N7:49 2 OTE B16:6/0 BND EOR
%   N7:49  FIC7030_MODE  "FIC7030 MODE 1=MAN 2=AUTO" %
%   B16:5/15  FY_7030_FIC7030_MAN  "FIC7030 MAN IND" %
%   B16:6/0  FY_7030_FIC7030_AUTO  "FIC7030 AUTO IND" %
% Rung: 271 %
SOR BST EQU N7:50 1 OTE B16:6/2 NXB EQU N7:50 2 OTE B16:6/3 BND EOR
%   N7:50  FIC7040_MODE  "FIC7040 MODE 1=MAN 2=AUTO" %
%   B16:6/2  FY_7040_FIC7040_MAN  "FIC7040 MAN IND" %
%   B16:6/3  FY_7040_FIC7040_AUTO  "FIC7040 AUTO IND" %
% Rung: 272 %
SOR BST EQU N7:51 1 OTE B16:6/5 NXB EQU N7:51 2 OTE B16:6/6 BND EOR
%   N7:51  LIC7030_MODE  "LIC7030 MODE 1=MAN 2=AUTO" %
%   B16:6/5  LY_7030_LIC7030_MAN  "LIC7030 MAN IND" %
%   B16:6/6  LY_7030_LIC7030_AUTO  "LIC7030 AUTO IND" %

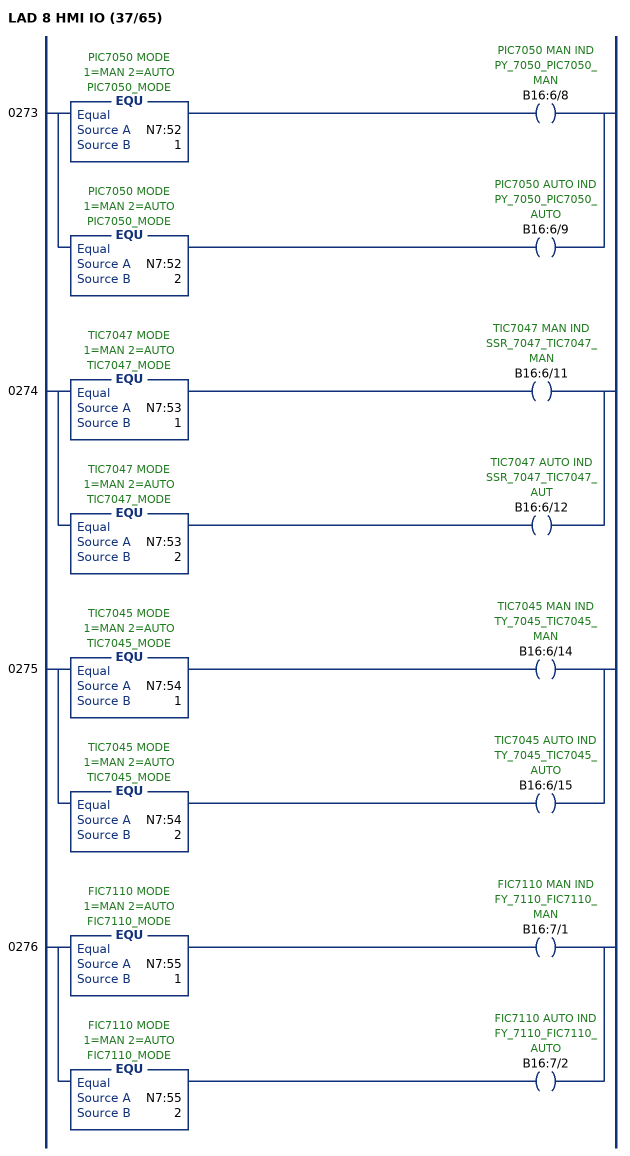
% Rung: 273 %
SOR BST EQU N7:52 1 OTE B16:6/8 NXB EQU N7:52 2 OTE B16:6/9 BND EOR
%   N7:52  PIC7050_MODE  "PIC7050 MODE 1=MAN 2=AUTO" %
%   B16:6/8  PY_7050_PIC7050_MAN  "PIC7050 MAN IND" %
%   B16:6/9  PY_7050_PIC7050_AUTO  "PIC7050 AUTO IND" %
% Rung: 274 %
SOR BST EQU N7:53 1 OTE B16:6/11 NXB EQU N7:53 2 OTE B16:6/12 BND EOR
%   N7:53  TIC7047_MODE  "TIC7047 MODE 1=MAN 2=AUTO" %
%   B16:6/11  SSR_7047_TIC7047_MAN  "TIC7047 MAN IND" %
%   B16:6/12  SSR_7047_TIC7047_AUT  "TIC7047 AUTO IND" %
% Rung: 275 %
SOR BST EQU N7:54 1 OTE B16:6/14 NXB EQU N7:54 2 OTE B16:6/15 BND EOR
%   N7:54  TIC7045_MODE  "TIC7045 MODE 1=MAN 2=AUTO" %
%   B16:6/14  TY_7045_TIC7045_MAN  "TIC7045 MAN IND" %
%   B16:6/15  TY_7045_TIC7045_AUTO  "TIC7045 AUTO IND" %
% Rung: 276 %
SOR BST EQU N7:55 1 OTE B16:7/1 NXB EQU N7:55 2 OTE B16:7/2 BND EOR
%   N7:55  FIC7110_MODE  "FIC7110 MODE 1=MAN 2=AUTO" %
%   B16:7/1  FY_7110_FIC7110_MAN  "FIC7110 MAN IND" %
%   B16:7/2  FY_7110_FIC7110_AUTO  "FIC7110 AUTO IND" %

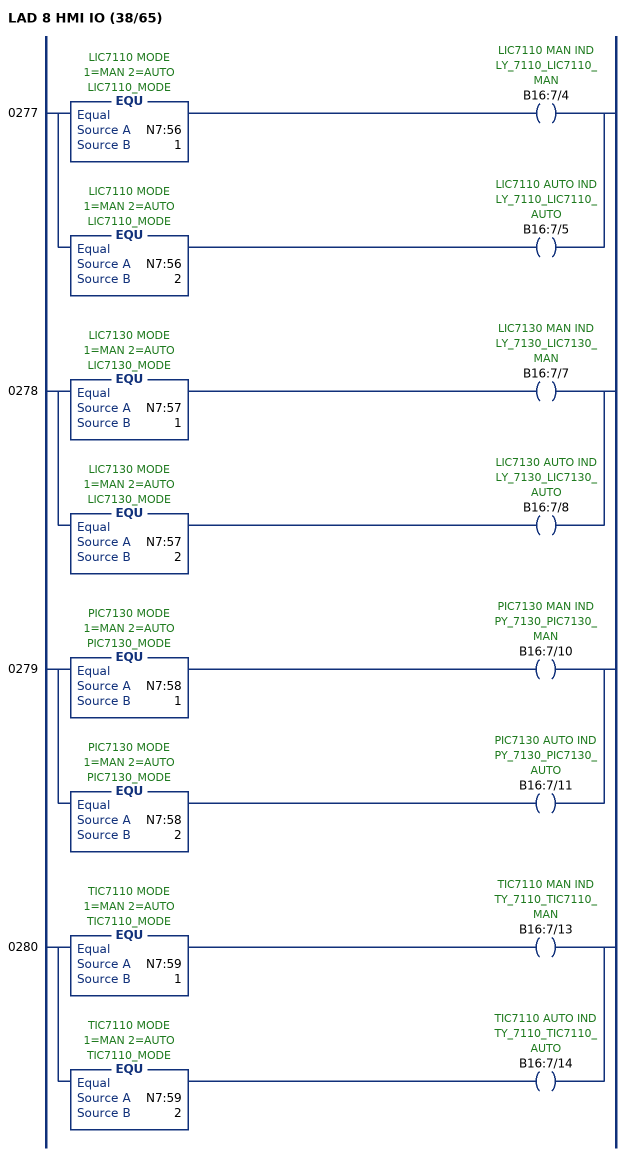
% Rung: 277 %
SOR BST EQU N7:56 1 OTE B16:7/4 NXB EQU N7:56 2 OTE B16:7/5 BND EOR
%   N7:56  LIC7110_MODE  "LIC7110 MODE 1=MAN 2=AUTO" %
%   B16:7/4  LY_7110_LIC7110_MAN  "LIC7110 MAN IND" %
%   B16:7/5  LY_7110_LIC7110_AUTO  "LIC7110 AUTO IND" %
% Rung: 278 %
SOR BST EQU N7:57 1 OTE B16:7/7 NXB EQU N7:57 2 OTE B16:7/8 BND EOR
%   N7:57  LIC7130_MODE  "LIC7130 MODE 1=MAN 2=AUTO" %
%   B16:7/7  LY_7130_LIC7130_MAN  "LIC7130 MAN IND" %
%   B16:7/8  LY_7130_LIC7130_AUTO  "LIC7130 AUTO IND" %
% Rung: 279 %
SOR BST EQU N7:58 1 OTE B16:7/10 NXB EQU N7:58 2 OTE B16:7/11 BND EOR
%   N7:58  PIC7130_MODE  "PIC7130 MODE 1=MAN 2=AUTO" %
%   B16:7/10  PY_7130_PIC7130_MAN  "PIC7130 MAN IND" %
%   B16:7/11  PY_7130_PIC7130_AUTO  "PIC7130 AUTO IND" %
% Rung: 280 %
SOR BST EQU N7:59 1 OTE B16:7/13 NXB EQU N7:59 2 OTE B16:7/14 BND EOR
%   N7:59  TIC7110_MODE  "TIC7110 MODE 1=MAN 2=AUTO" %
%   B16:7/13  TY_7110_TIC7110_MAN  "TIC7110 MAN IND" %
%   B16:7/14  TY_7110_TIC7110_AUTO  "TIC7110 AUTO IND" %

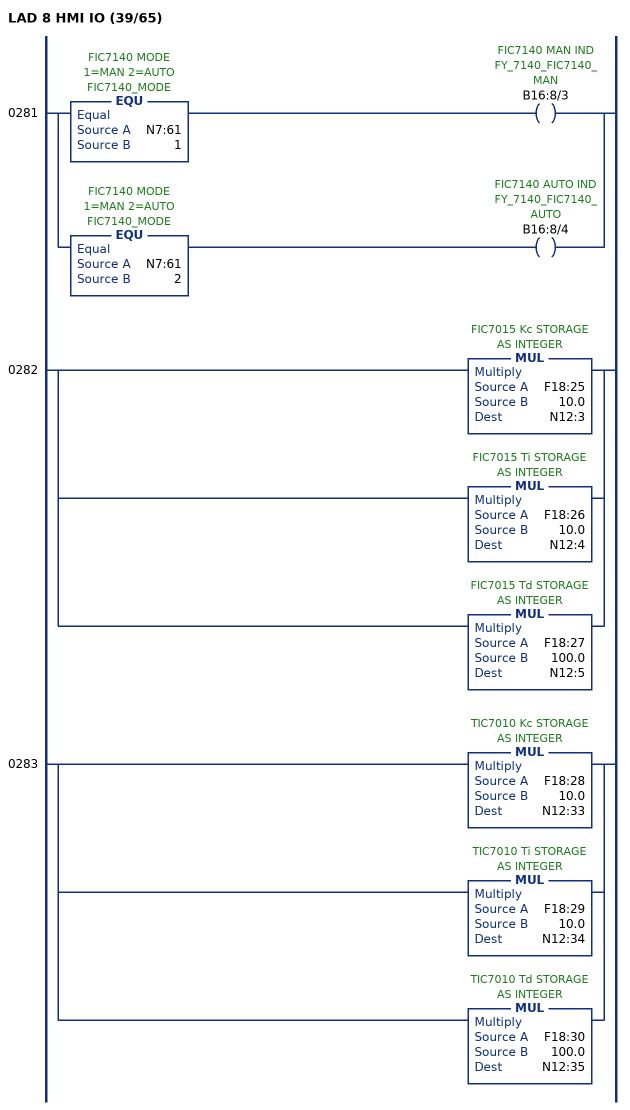
% Rung: 281 %
SOR BST EQU N7:61 1 OTE B16:8/3 NXB EQU N7:61 2 OTE B16:8/4 BND EOR
%   N7:61  FIC7140_MODE  "FIC7140 MODE 1=MAN 2=AUTO" %
%   B16:8/3  FY_7140_FIC7140_MAN  "FIC7140 MAN IND" %
%   B16:8/4  FY_7140_FIC7140_AUTO  "FIC7140 AUTO IND" %
% Rung: 282 %
SOR BST MUL F18:25 10.0 N12:3 NXB MUL F18:26 10.0 N12:4 NXB MUL F18:27 100.0 N12:5 BND EOR
%   F18:25  FIC7015_KC  "FIC7015 Kc" %
%   N12:3  "FIC7015 Kc STORAGE AS INTEGER" %
%   F18:26  FIC7015_TI  "FIC7015 Ti" %
%   N12:4  "FIC7015 Ti STORAGE AS INTEGER" %
%   F18:27  FIC7015_TD  "FIC7015 Td" %
%   N12:5  "FIC7015 Td STORAGE AS INTEGER" %
% Rung: 283 %
SOR BST MUL F18:28 10.0 N12:33 NXB MUL F18:29 10.0 N12:34 NXB MUL F18:30 100.0 N12:35 BND EOR
%   F18:28  TIC7010_KC  "TIC7010 Kc" %
%   N12:33  "TIC7010 Kc STORAGE AS INTEGER" %
%   F18:29  TIC7010_TI  "TIC7010 Ti" %
%   N12:34  "TIC7010 Ti STORAGE AS INTEGER" %
%   F18:30  TIC7010_TD  "TIC7010_Td" %
%   N12:35  "TIC7010 Td STORAGE AS INTEGER" %

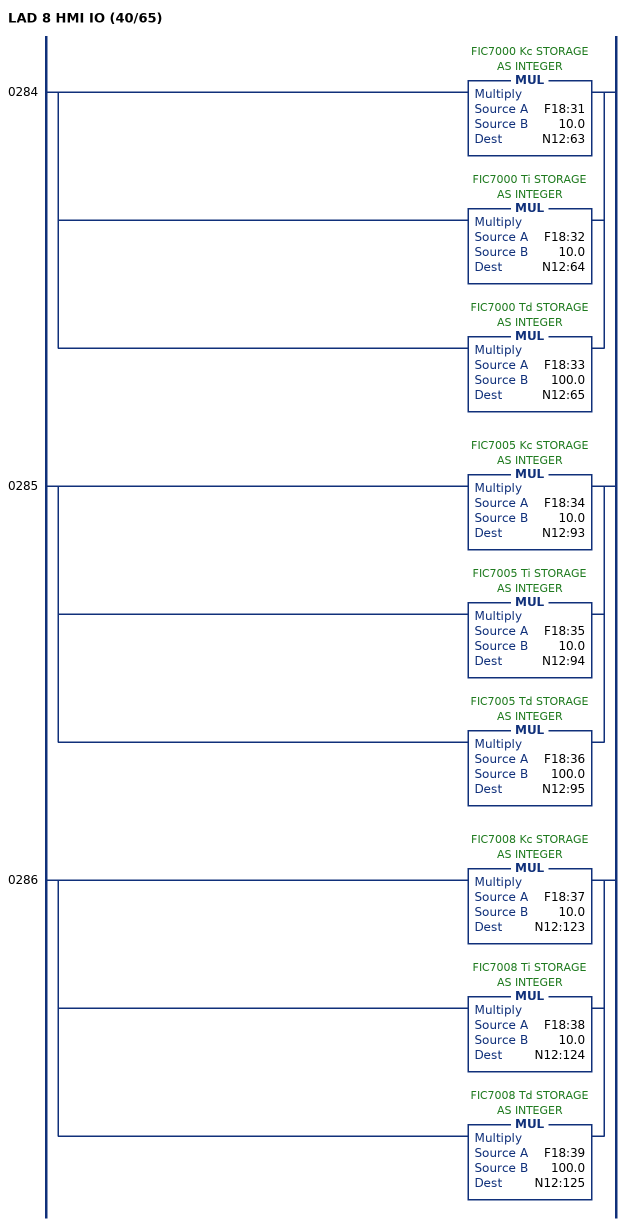
% Rung: 284 %
SOR BST MUL F18:31 10.0 N12:63 NXB MUL F18:32 10.0 N12:64 NXB MUL F18:33 100.0 N12:65 BND EOR
%   F18:31  FIC7000_KC  "FIC7000 Kc" %
%   N12:63  "FIC7000 Kc STORAGE AS INTEGER" %
%   F18:32  FIC7000_TI  "FIC7000 Ti" %
%   N12:64  "FIC7000 Ti STORAGE AS INTEGER" %
%   F18:33  FIC7000_TD  "FIC7000 Td" %
%   N12:65  "FIC7000 Td STORAGE AS INTEGER" %
% Rung: 285 %
SOR BST MUL F18:34 10.0 N12:93 NXB MUL F18:35 10.0 N12:94 NXB MUL F18:36 100.0 N12:95 BND EOR
%   F18:34  FIC7005_KC  "FIC7005 Kc" %
%   N12:93  "FIC7005 Kc STORAGE AS INTEGER" %
%   F18:35  FIC7005_TI  "FIC7005 Ti" %
%   N12:94  "FIC7005 Ti STORAGE AS INTEGER" %
%   F18:36  FIC7005_TD  "FIC7005 Td" %
%   N12:95  "FIC7005 Td STORAGE AS INTEGER" %
% Rung: 286 %
SOR BST MUL F18:37 10.0 N12:123 NXB MUL F18:38 10.0 N12:124 NXB MUL F18:39 100.0 N12:125 BND EOR
%   F18:37  FIC7008_KC  "FIC7008 Kc" %
%   N12:123  "FIC7008 Kc STORAGE AS INTEGER" %
%   F18:38  FIC7008_TI  "FIC7008 Ti" %
%   N12:124  "FIC7008 Ti STORAGE AS INTEGER" %
%   F18:39  FIC7008_TD  "FIC7008 Td" %
%   N12:125  "FIC7008 Td STORAGE AS INTEGER" %

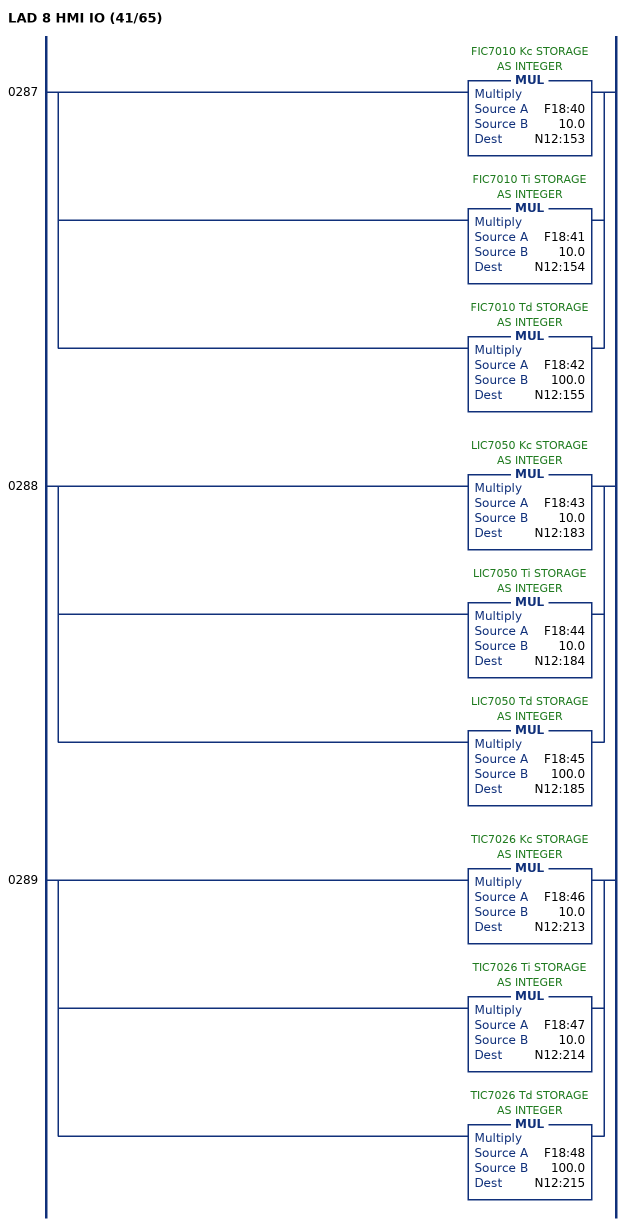
% Rung: 287 %
SOR BST MUL F18:40 10.0 N12:153 NXB MUL F18:41 10.0 N12:154 NXB MUL F18:42 100.0 N12:155 BND EOR
%   F18:40  FIC7010_KC  "FIC7010 Kc" %
%   N12:153  "FIC7010 Kc STORAGE AS INTEGER" %
%   F18:41  FIC7010_TI  "FIC7010 Ti" %
%   N12:154  "FIC7010 Ti STORAGE AS INTEGER" %
%   F18:42  FIC7010_TD  "FIC7010_Td" %
%   N12:155  "FIC7010 Td STORAGE AS INTEGER" %
% Rung: 288 %
SOR BST MUL F18:43 10.0 N12:183 NXB MUL F18:44 10.0 N12:184 NXB MUL F18:45 100.0 N12:185 BND EOR
%   F18:43  LIC7050_KC  "LIC7050 Kc" %
%   N12:183  "LIC7050 Kc STORAGE AS INTEGER" %
%   F18:44  LIC7050_TI  "LIC7050 Ti" %
%   N12:184  "LIC7050 Ti STORAGE AS INTEGER" %
%   F18:45  LIC7050_TD  "LIC7050 Td" %
%   N12:185  "LIC7050 Td STORAGE AS INTEGER" %
% Rung: 289 %
SOR BST MUL F18:46 10.0 N12:213 NXB MUL F18:47 10.0 N12:214 NXB MUL F18:48 100.0 N12:215 BND EOR
%   F18:46  TIC7026_KC  "TIC7026 Kc" %
%   N12:213  "TIC7026 Kc STORAGE AS INTEGER" %
%   F18:47  TIC7026_TI  "TIC7026 Ti" %
%   N12:214  "TIC7026 Ti STORAGE AS INTEGER" %
%   F18:48  TIC7026_TD  "TIC7026 Td" %
%   N12:215  "TIC7026 Td STORAGE AS INTEGER" %

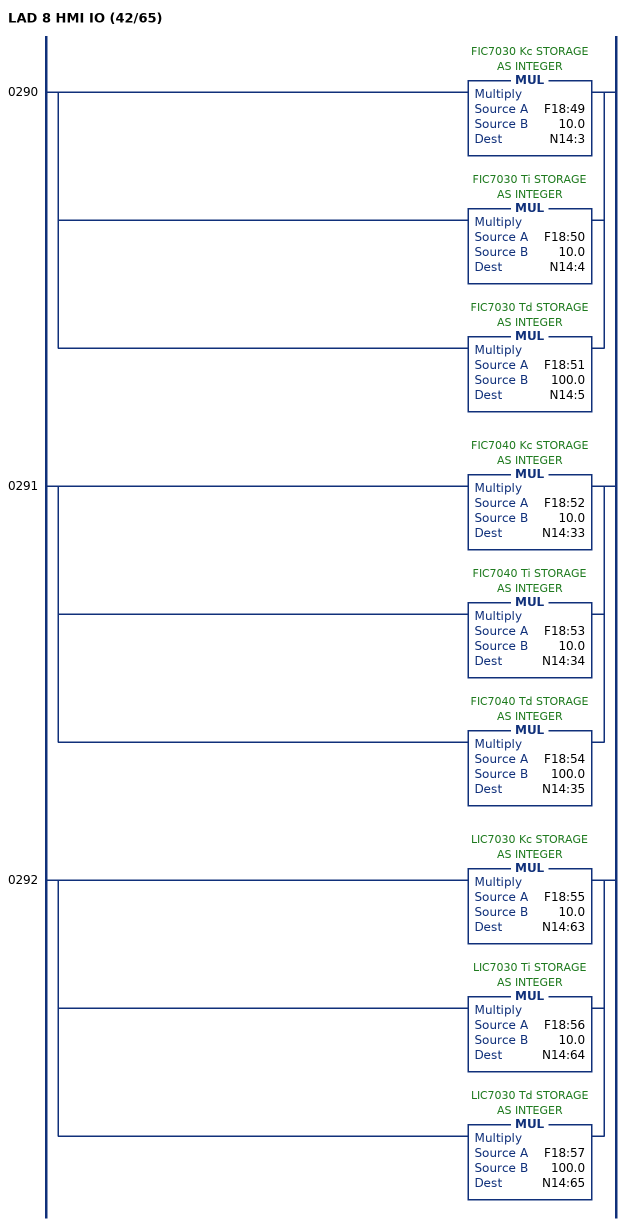
% Rung: 290 %
SOR BST MUL F18:49 10.0 N14:3 NXB MUL F18:50 10.0 N14:4 NXB MUL F18:51 100.0 N14:5 BND EOR
%   F18:49  FIC7030_KC  "FIC7030 Kc" %
%   N14:3  "FIC7030 Kc STORAGE AS INTEGER" %
%   F18:50  FIC7030_TI  "FIC7030 Ti" %
%   N14:4  "FIC7030 Ti STORAGE AS INTEGER" %
%   F18:51  FIC7030_TD  "FIC7030 Td" %
%   N14:5  "FIC7030 Td STORAGE AS INTEGER" %
% Rung: 291 %
SOR BST MUL F18:52 10.0 N14:33 NXB MUL F18:53 10.0 N14:34 NXB MUL F18:54 100.0 N14:35 BND EOR
%   F18:52  FIC7040_KC  "FIC7040 Kc" %
%   N14:33  "FIC7040 Kc STORAGE AS INTEGER" %
%   F18:53  FIC7040_TI  "FIC7040 Ti" %
%   N14:34  "FIC7040 Ti STORAGE AS INTEGER" %
%   F18:54  FIC7040_TD  "FIC7040 Td" %
%   N14:35  "FIC7040 Td STORAGE AS INTEGER" %
% Rung: 292 %
SOR BST MUL F18:55 10.0 N14:63 NXB MUL F18:56 10.0 N14:64 NXB MUL F18:57 100.0 N14:65 BND EOR
%   F18:55  LIC7030_KC  "LIC7030 Kc" %
%   N14:63  "LIC7030 Kc STORAGE AS INTEGER" %
%   F18:56  LIC7030_TI  "LIC7030 Ti" %
%   N14:64  "LIC7030 Ti STORAGE AS INTEGER" %
%   F18:57  LIC7030_TD  "LIC7030 Td" %
%   N14:65  "LIC7030 Td STORAGE AS INTEGER" %

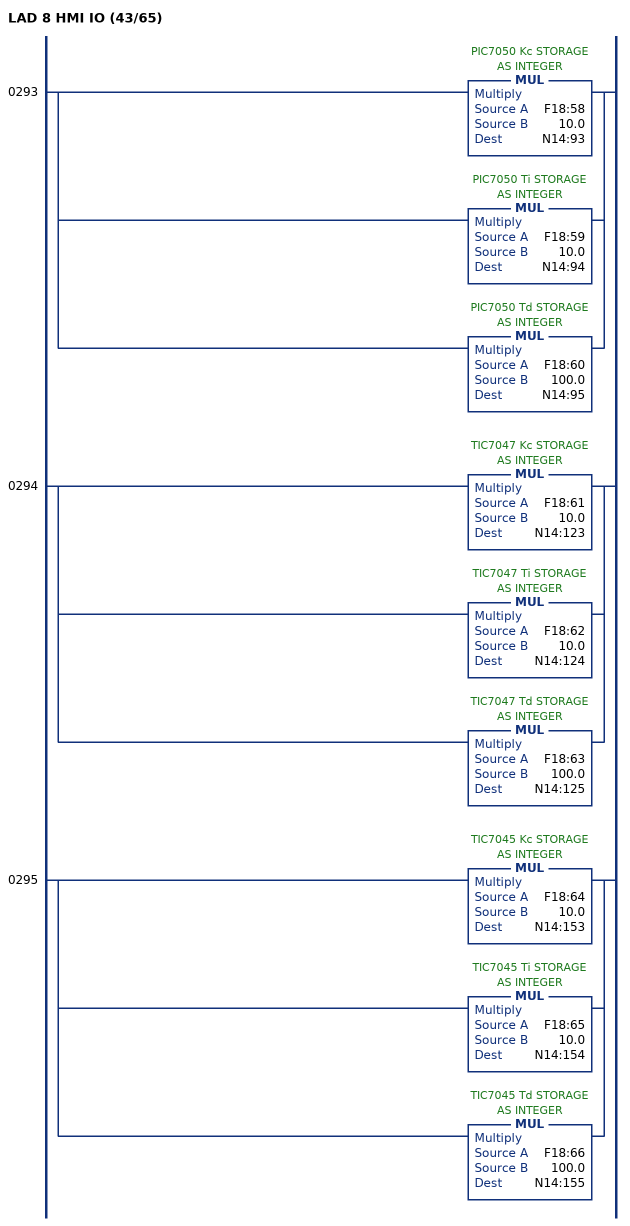
% Rung: 293 %
SOR BST MUL F18:58 10.0 N14:93 NXB MUL F18:59 10.0 N14:94 NXB MUL F18:60 100.0 N14:95 BND EOR
%   F18:58  PIC7050_KC  "PIC7050 Kc" %
%   N14:93  "PIC7050 Kc STORAGE AS INTEGER" %
%   F18:59  PIC7050_TI  "PIC7050 Ti" %
%   N14:94  "PIC7050 Ti STORAGE AS INTEGER" %
%   F18:60  PIC7050_TD  "PIC7050 Td" %
%   N14:95  "PIC7050 Td STORAGE AS INTEGER" %
% Rung: 294 %
SOR BST MUL F18:61 10.0 N14:123 NXB MUL F18:62 10.0 N14:124 NXB MUL F18:63 100.0 N14:125 BND EOR
%   F18:61  TIC7047_KC  "TIC7047 Kc" %
%   N14:123  "TIC7047 Kc STORAGE AS INTEGER" %
%   F18:62  TIC7047_TI  "TIC7047 Ti" %
%   N14:124  "TIC7047 Ti STORAGE AS INTEGER" %
%   F18:63  TIC7047_TD  "TIC7047 Td" %
%   N14:125  "TIC7047 Td STORAGE AS INTEGER" %
% Rung: 295 %
SOR BST MUL F18:64 10.0 N14:153 NXB MUL F18:65 10.0 N14:154 NXB MUL F18:66 100.0 N14:155 BND EOR
%   F18:64  TIC7045_KC  "TIC7045 Kc" %
%   N14:153  "TIC7045 Kc STORAGE AS INTEGER" %
%   F18:65  TIC7045_TI  "TIC7045 Ti" %
%   N14:154  "TIC7045 Ti STORAGE AS INTEGER" %
%   F18:66  TIC7045_TD  "TIC7045 Td" %
%   N14:155  "TIC7045 Td STORAGE AS INTEGER" %

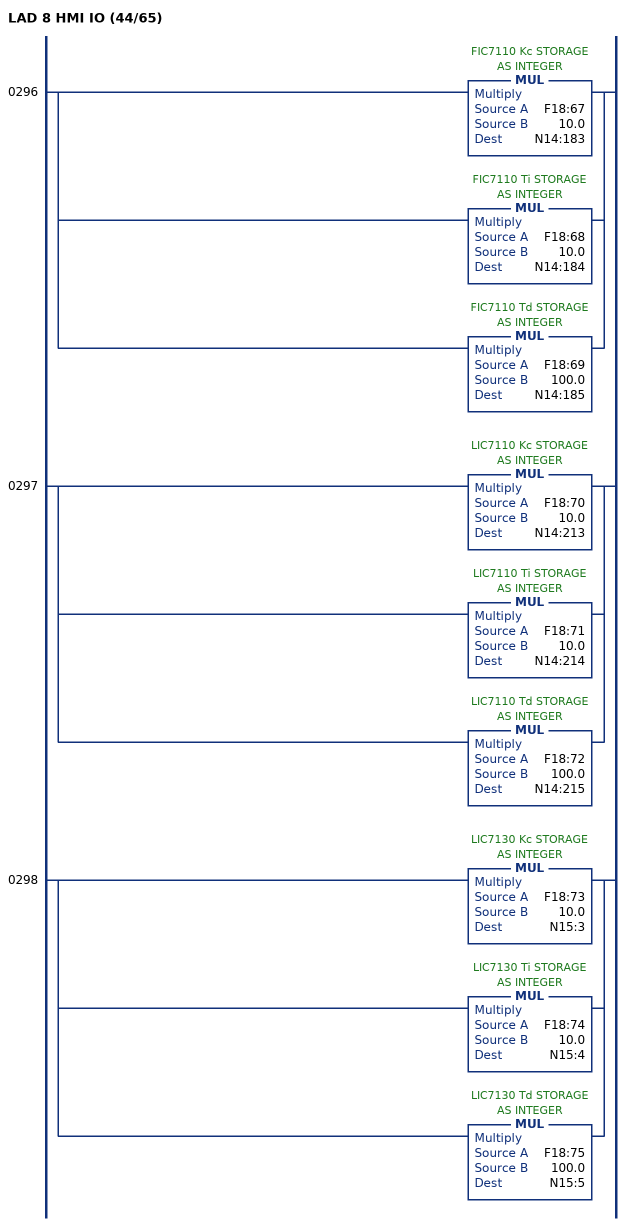
% Rung: 296 %
SOR BST MUL F18:67 10.0 N14:183 NXB MUL F18:68 10.0 N14:184 NXB MUL F18:69 100.0 N14:185 BND EOR
%   F18:67  FIC7110_KC  "FIC7110 Kc" %
%   N14:183  "FIC7110 Kc STORAGE AS INTEGER" %
%   F18:68  FIC7110_TI  "FIC7110 Ti" %
%   N14:184  "FIC7110 Ti STORAGE AS INTEGER" %
%   F18:69  FIC7110_TD  "FIC7110 Td" %
%   N14:185  "FIC7110 Td STORAGE AS INTEGER" %
% Rung: 297 %
SOR BST MUL F18:70 10.0 N14:213 NXB MUL F18:71 10.0 N14:214 NXB MUL F18:72 100.0 N14:215 BND EOR
%   F18:70  LIC7110_KC  "LIC7110 Kc" %
%   N14:213  "LIC7110 Kc STORAGE AS INTEGER" %
%   F18:71  LIC7110_TI  "LIC7110 Ti" %
%   N14:214  "LIC7110 Ti STORAGE AS INTEGER" %
%   F18:72  LIC7110_TD  "LIC7110 Td" %
%   N14:215  "LIC7110 Td STORAGE AS INTEGER" %
% Rung: 298 %
SOR BST MUL F18:73 10.0 N15:3 NXB MUL F18:74 10.0 N15:4 NXB MUL F18:75 100.0 N15:5 BND EOR
%   F18:73  LIC7130_KC  "LIC7130 Kc" %
%   N15:3  "LIC7130 Kc STORAGE AS INTEGER" %
%   F18:74  LIC7130_TI  "LIC7130 Ti" %
%   N15:4  "LIC7130 Ti STORAGE AS INTEGER" %
%   F18:75  LIC7130_TD  "LIC7130 Td" %
%   N15:5  "LIC7130 Td STORAGE AS INTEGER" %

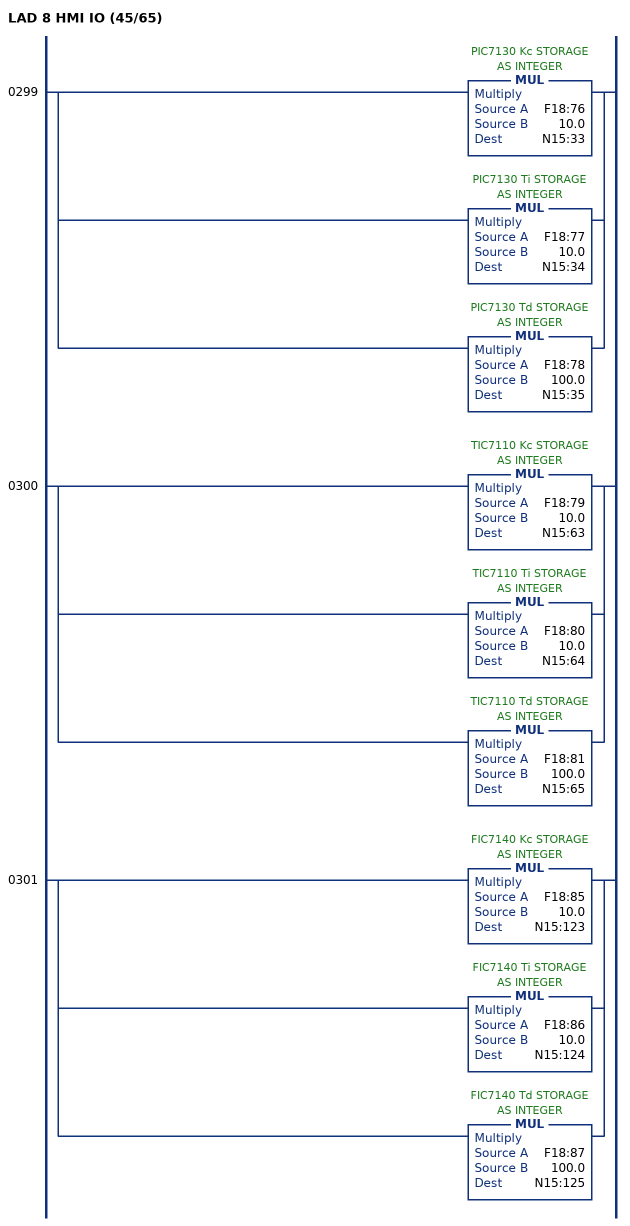
% Rung: 299 %
SOR BST MUL F18:76 10.0 N15:33 NXB MUL F18:77 10.0 N15:34 NXB MUL F18:78 100.0 N15:35 BND EOR
%   F18:76  PIC7130_KC  "PIC7130 Kc" %
%   N15:33  "PIC7130 Kc STORAGE AS INTEGER" %
%   F18:77  PIC7130_TI  "PIC7130 Ti" %
%   N15:34  "PIC7130 Ti STORAGE AS INTEGER" %
%   F18:78  PIC7130_TD  "PIC7130 Td" %
%   N15:35  "PIC7130 Td STORAGE AS INTEGER" %
% Rung: 300 %
SOR BST MUL F18:79 10.0 N15:63 NXB MUL F18:80 10.0 N15:64 NXB MUL F18:81 100.0 N15:65 BND EOR
%   F18:79  TIC7110_KC  "TIC7110 Kc" %
%   N15:63  "TIC7110 Kc STORAGE AS INTEGER" %
%   F18:80  TIC7110_TI  "TIC7110 Ti" %
%   N15:64  "TIC7110 Ti STORAGE AS INTEGER" %
%   F18:81  TIC7110_TD  "TIC7110 Td" %
%   N15:65  "TIC7110 Td STORAGE AS INTEGER" %
% Rung: 301 %
SOR BST MUL F18:85 10.0 N15:123 NXB MUL F18:86 10.0 N15:124 NXB MUL F18:87 100.0 N15:125 BND EOR
%   F18:85  FIC7140_KC  "FIC7140 Kc" %
%   N15:123  "FIC7140 Kc STORAGE AS INTEGER" %
%   F18:86  FIC7140_TI  "FIC7140 Ti" %
%   N15:124  "FIC7140 Ti STORAGE AS INTEGER" %
%   F18:87  FIC7140_TD  "FIC7140 Td" %
%   N15:125  "FIC7140 Td STORAGE AS INTEGER" %

